// TIA Portal V20 export
FUNCTION_BLOCK "CallEquipment"   // FB72, LAD
TITLE = CallEquipment
// This block includes all general functions, checks and logik that is needed in the entire unit. E.g. general releases and system wide functionalities like air, pressure and power handling as well as general reaction to events.
// stored: IsIECCheckEnabled true, MemoryReserve 100, Namespace Unit1.Em8, SetENOAutomatically true
   VAR_INPUT
      ZoneOperationEnable { ExternalWritable := 'False'} : "LWONIK_typeSafetyZoneManualOperation";
   END_VAR
   VAR_IN_OUT
      unitStatus : "LAF_typeUnitStatus";   // Current unit status o be used in this EM
      emFeedback : "LUC_typeEmFeedback";   // Feedback of the EM to the Unit
      unitAlarmDB : "LAF_typeAlarms";   // Summarized EM Alarms for the Unit
   END_VAR
   VAR
      InstHipotThicknessSequence { ExternalWritable := 'False'} : "Unit1.Em8.Sequence_1_HipotThickness";
      InstHipotThicknessRnRSequence { S7_SetPoint := 'True'} : "Unit1.Em8.Sequence_10_GuageRnR";
      instHipotThicknessHomeJob1 { ExternalWritable := 'False'} : "LAF_SelectJob";
      instHipotThicknessLoadJob2 { ExternalWritable := 'False'} : "LAF_SelectJob";
      instHipotThicknessInspectionJob3 { ExternalWritable := 'False'} : "LAF_SelectJob";
      instHipotThicknessUnloadJob4 { ExternalWritable := 'False'} : "LAF_SelectJob";
      instGRnR_HipotThicknessLoad_Job2 { S7_SetPoint := 'True'} : "LAF_SelectJob";
      instGRnR_HipotThicknessInspection_Job3 { S7_SetPoint := 'True'} : "LAF_SelectJob";
      instGRnR_HipotThicknessUnload_Job4 { S7_SetPoint := 'True'} : "LAF_SelectJob";
      instCmHipotThicknessSafetyPin { ExternalWritable := 'False'} : "LBC_DigitalSignalCn";
      instCmHipotThicknessJRDetect { ExternalWritable := 'False'} : "LBC_DigitalSignalCn";
      instCmThicknessAxisZ { ExternalWritable := 'False'} : "LBC_Axis64Pos_TecPlcCn";
      instCmHipotThinknessStageLiftFrontUpDown { ExternalWritable := 'False'} : "LBC_TwoWayActuatorCn";
      instCmHipotThinknessStageLiftRearUpDown { ExternalWritable := 'False'} : "LBC_TwoWayActuatorCn";
      instCmHipotTabContactorBwdFwd { ExternalWritable := 'False'} : "LBC_TwoWayActuatorCn";
      instCmHipotTabContactorLeftOpenClose { ExternalWritable := 'False'} : "LBC_TwoWayActuatorCn";
      instCmHipotTabContactorRightOpenClose { ExternalWritable := 'False'} : "LBC_TwoWayActuatorCn";
      instCmHipotThinknessStageLiftAllUpDown { ExternalWritable := 'False'} : "LBC_TwoWayActuatorCn";
      instCmHipotControl { ExternalWritable := 'False'} : "LER_IRCheck_BT5525";
      instCmThicknessControl { ExternalWritable := 'False'} : "LER_Thickness";
      instCmHipotThicknessServoPress { ExternalWritable := 'False'} : "LER_ServoPress";
      instInterlockThicknessAxisZ { ExternalWritable := 'False'} : "LER_Axis64Pos_InterlockSummary";
      instLDrv701ControlThicknessAxisZ { ExternalWritable := 'False'} : "LDrvSafe_SinaTlg701Control";   // Drive Telegram Function Library
      instLDrv701StatusThicknessAxisZ { ExternalWritable := 'False'} : "LDrvSafe_SinaTlg701Status";   // Drive Telegram Function Library
      instHipotThicknessPressHistory { ExternalWritable := 'False'} : "LER_ServoPressHistory";
      instHipotHistory { ExternalWritable := 'False'} : "LER_hipotHistory";
      instThicknessHistory { ExternalWritable := 'False'} : "LER_thicknessHistory";
      instManageAlarms { ExternalWritable := 'False'} : "LAF_ManageAlarms";
      instEventsPFE { ExternalWritable := 'False'} : "Unit1.Em8.EventsPFE";
      statUnitStatus { ExternalWritable := 'False'} : "LAF_typeUnitStatus";   // Unit Status that is used in this project
      statSlmStatus { ExternalWritable := 'False'} : Struct
         running : Bool;
         powerOff : Bool;
      END_STRUCT;
      statAllBrakeTest { ExternalWritable := 'False'} : "LER_typeBrakeTestUnitCommands";
      statPartData { ExternalWritable := 'False'} : "LER_typePartData";
      statDataDelete { ExternalWritable := 'False'} : "LER_typePartData";
      statHistoryDeleteData_press { ExternalWritable := 'False'} : "LER_typeServoPressHistory";
      statHistoryDeleteData_hipot { ExternalWritable := 'False'} : "LER_typeHipotHistory";
      statHistoryDeleteData_thickness { ExternalWritable := 'False'} : "LER_typeThicknessHistory";
      "statHistoryDeleteData_thicknessR&R" { ExternalWritable := 'False'} : "LER_typeThicknessHistory_R&R";
      statRoutingOk { ExternalWritable := 'False'} : Array[0..99] of Bool;
      statRoutingNok { ExternalWritable := 'False'} : Array[0..99] of Bool;
      statTonTime { ExternalWritable := 'False'} : Array[0..999] of TON_TIME;
      statTofTime { ExternalWritable := 'False'} : Array[0..9] of TOF_TIME;
      statPulse { ExternalWritable := 'False'} : Array[0..999] of Bool;
      statGaugeRnR { ExternalWritable := 'False'} : Struct
         currentCount : Int;
         processCount : Int;
         Ongoing : Bool;
         Complete : Bool;
      END_STRUCT;
      statEnableManualCmds { ExternalWritable := 'False'} : Bool;
      statNomalMode { ExternalWritable := 'False'} : Bool;
      "*** Interlock Axis ***" : Bool;
      ThicknessAxisZ_Jog { S7_SetPoint := 'True'} : Array[0..2] of "LER_Axis_Jog";
      ThicknessAxisZ_interlock { S7_SetPoint := 'True'} : Array[0..10] of "LER_Axis_Absolute";
      ThicknessAxisZ_IntPos : Array[0..9] of Struct
         "Int" : Array[1..10] of Bool;
      END_STRUCT;
      ThicknessAxisZ_IntHome : Array[0..9] of Bool;
      ThicknessAxisZ_PosAbsolute : Array[0..10] of Bool;
      ThicknessAxisZ_Home { S7_SetPoint := 'True'} : "LER_Axis_Homing";
      "*** Interlock TwoWay ***" { S7_SetPoint := 'True'} : "LER_Axis_Homing";
      instCmHipotThinknessStageLiftFrontUpDownInterlock { S7_SetPoint := 'True'} : Array[0..2] of "LER_Actuator";
      instCmHipotThinknessStageLiftRearUpDownInterlock { S7_SetPoint := 'True'} : Array[0..2] of "LER_Actuator";
      instCmHipotTabContactorBwdFwdInterlock { S7_SetPoint := 'True'} : Array[0..2] of "LER_Actuator";
      instCmHipotTabContactorLeftOpenCloseInterlock { S7_SetPoint := 'True'} : Array[0..2] of "LER_Actuator";
      instCmHipotTabContactorRightOpenCloseInterlock { S7_SetPoint := 'True'} : Array[0..2] of "LER_Actuator";
      instCmHipotThinknessStageLiftAllUpDownInterlock { S7_SetPoint := 'True'} : Array[0..2] of "LER_Actuator";
      HipotThinknessStageLiftFrontUpDown_Inpos : Array[0..2] of Struct
         "Int" : Array[1..10] of Bool;
      END_STRUCT;
      HipotThinknessStageLiftRearUpDown_Inpos : Array[0..2] of Struct
         "Int" : Array[1..10] of Bool;
      END_STRUCT;
      HipotTabContactorBwdFwd_Inpos : Array[0..2] of Struct
         "Int" : Array[1..10] of Bool;
      END_STRUCT;
      HipotTabContactorLeftOpenClose_Inpos : Array[0..2] of Struct
         "Int" : Array[1..10] of Bool;
      END_STRUCT;
      HipotTabContactorRightOpenClose_Inpos : Array[0..2] of Struct
         "Int" : Array[1..10] of Bool;
      END_STRUCT;
      HipotThinknessStageLiftAllUpDown_Inpos : Array[0..2] of Struct
         "Int" : Array[1..10] of Bool;
      END_STRUCT;
      citi_Ptrig : Array[0..20] of Bool;
      citiTon : Array[0..20] of TON_TIME;
      citi : Time;
      citiTest : Array[0..20] of Bool;
      instPFERecipe { S7_SetPoint := 'True'} : "Unit1.Em8.EventsPFE_Recipe";
   END_VAR
   VAR_TEMP
      tempRET_VAL : Array[0..99] of Int;
      tempScInProduction : Bool;   // Mode Production and StateComplete
      tempScNoProduction : Bool;   // Mode Manual and StateComplete
      tempPlaceReq : Bool;   // Request placing to TRPnPRight
      tempInspecReq : Bool;
      tempPickReq : Bool;   // Request Pick to TRPnPRight
   END_VAR
   VAR CONSTANT
      delayTime : Time := T#3s;
      TRUE : Bool := TRUE;
      FALSE : Bool;
      NO_JOB : DInt;
      MIN_POSITION_NUMBER : SInt;
      INIT_POSITION_NUMBER : SInt := -1;
   END_VAR
   VAR_TEMP   // added for the SCL form of the ladder/FBD networks
      _w1 : Bool;
      _w2 : Bool;
      _w3 : Bool;
      _w4 : Bool;
      _w5 : Bool;
      _w6 : Bool;
      _w7 : Bool;
      _w8 : Bool;
      _w9 : Bool;
      _w10 : Bool;
      _w11 : Bool;
      _w12 : Bool;
   END_VAR
BEGIN

REGION Network 1: BLOCK INFO HEADER
   // (company) / (C) Copyright (year)
   // ---------------------------------------------------------------------------------
   // Title:                             (Title of this block)
   // Comment/Function: (that is implemented in the block)
   // Library/Family:           (that the source is dedicated to)
   // Author:                        (department / person in charge / contact)
   // Target System:          (test system with FW version)
   // Engineering:              TIA Portal (SW version)
   // Restrictions:               (OB types, etc.)
   // Requirements:           (hardware, technological package, etc.)
   // ---------------------------------------------------------------------------------
   // Change log table:
   // Version          | Date             | Signature      | Expert in charge  | Changes applied ------------------------|----------------------|-------------------------|--------------------------------|-----------------------
   // 001.000.000 | yyyy-mm-dd | 0x00000000 | (name of expert) | First released version
END_REGION

REGION Network 2: DESCRIPTION
   // This is a template block provided by the Automation Framework. It can be used to create an own project.
   // The Block Info Header is prepared to put in your own data.
   // Description of the block could be added here and the docu created by Code2Docu.
END_REGION

REGION Network 3: Simulation
   // If simulation is active on a global level, inherit this status and set simulation active in this unit also. Information is written to DB ControlNodes, from where it is distributed to the equipmemt modules.
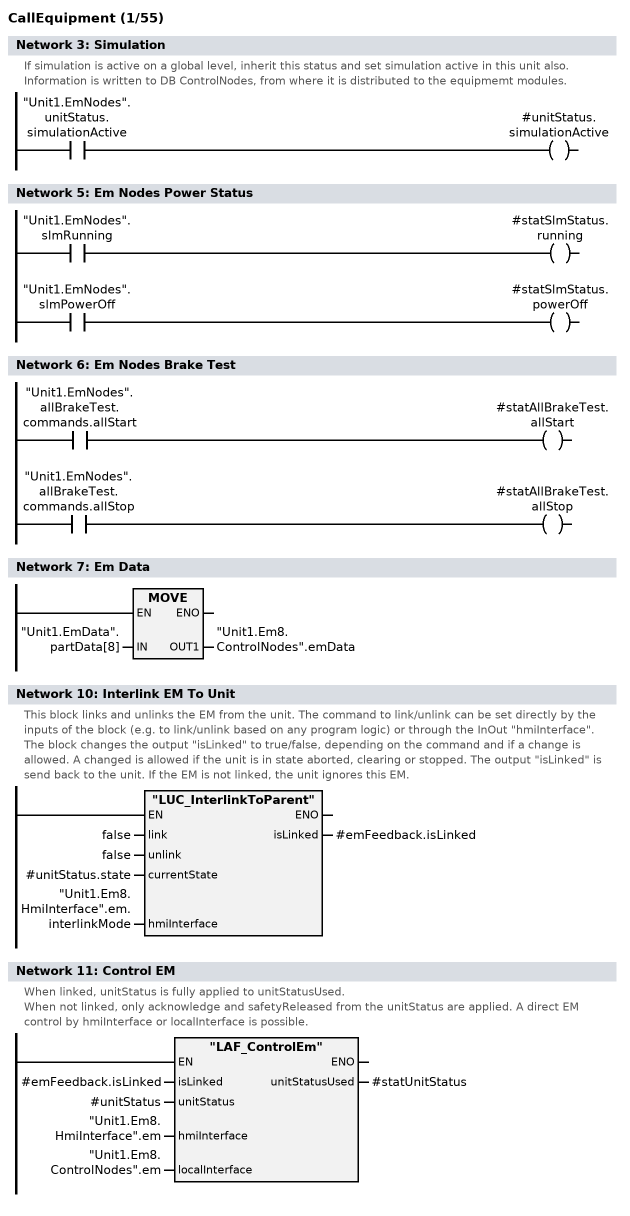
   RUNG wire#powerrail
      Contact( "Unit1.EmNodes".unitStatus.simulationActive )
      Coil( #unitStatus.simulationActive )
   END_RUNG
   // the same network as SCL:
   #unitStatus.simulationActive := "Unit1.EmNodes".unitStatus.simulationActive;
END_REGION

REGION Network 4: ******************** Unit Input ********************
END_REGION

REGION Network 5: Em Nodes Power Status
   RUNG wire#powerrail
      Contact( "Unit1.EmNodes".slmRunning )
      Coil( #statSlmStatus.running )
   END_RUNG
   RUNG wire#powerrail
      Contact( "Unit1.EmNodes".slmPowerOff )
      Coil( #statSlmStatus.powerOff )
   END_RUNG
   // the same network as SCL:
   #statSlmStatus.running := "Unit1.EmNodes".slmRunning;
   #statSlmStatus.powerOff := "Unit1.EmNodes".slmPowerOff;
END_REGION

REGION Network 6: Em Nodes Brake Test
   RUNG wire#powerrail
      Contact( "Unit1.EmNodes".allBrakeTest.commands.allStart )
      Coil( #statAllBrakeTest.allStart )
   END_RUNG
   RUNG wire#powerrail
      Contact( "Unit1.EmNodes".allBrakeTest.commands.allStop )
      Coil( #statAllBrakeTest.allStop )
   END_RUNG
   // the same network as SCL:
   #statAllBrakeTest.allStart := "Unit1.EmNodes".allBrakeTest.commands.allStart;
   #statAllBrakeTest.allStop := "Unit1.EmNodes".allBrakeTest.commands.allStop;
END_REGION

REGION Network 7: Em Data
   RUNG wire#powerrail
      Move(in := "Unit1.EmData".partData[8], out1 => "Unit1.Em8.ControlNodes".emData)
   END_RUNG
   // the same network as SCL:
   "Unit1.Em8.ControlNodes".emData := "Unit1.EmData".partData[8];
END_REGION

REGION Network 9: ******************** Equipment Control ********************
END_REGION

REGION Network 10: Interlink EM To Unit
   // This block links and unlinks the EM from the unit. The command to link/unlink can be set directly by the inputs of the block (e.g. to link/unlink based on any program logic) or through the InOut "hmiInterface". The block changes the output "isLinked" to true/false, depending on the command and if a change is allowed. A changed is allowed if the unit is in state aborted, clearing or stopped. The output "isLinked" is send back to the unit. If the EM is not linked, the unit ignores this EM.
   RUNG wire#powerrail
      "LUC_InterlinkToParent"(link := false, unlink := false, currentState := #unitStatus.state, hmiInterface := "Unit1.Em8.HmiInterface".em.interlinkMode, isLinked => #emFeedback.isLinked)
   END_RUNG
   // the same network as SCL:
   "LUC_InterlinkToParent"(link := false,
                           unlink := false,
                           currentState := #unitStatus.state,
                           hmiInterface := "Unit1.Em8.HmiInterface".em.interlinkMode,
                           isLinked => #emFeedback.isLinked);
END_REGION

REGION Network 11: Control EM
   // When linked, unitStatus is fully applied to unitStatusUsed.
   // When not linked, only acknowledge and safetyReleased from the unitStatus are applied. A direct EM control by hmiInterface or localInterface is possible.
   RUNG wire#powerrail
      "LAF_ControlEm"(isLinked := #emFeedback.isLinked, unitStatus := #unitStatus, hmiInterface := "Unit1.Em8.HmiInterface".em, localInterface := "Unit1.Em8.ControlNodes".em, unitStatusUsed => #statUnitStatus)
   END_RUNG
   // the same network as SCL:
   "LAF_ControlEm"(isLinked := #emFeedback.isLinked,
                   unitStatus := #unitStatus,
                   hmiInterface := "Unit1.Em8.HmiInterface".em,
                   localInterface := "Unit1.Em8.ControlNodes".em,
                   unitStatusUsed => #statUnitStatus);
END_REGION

REGION Network 12: EnableManualCmds
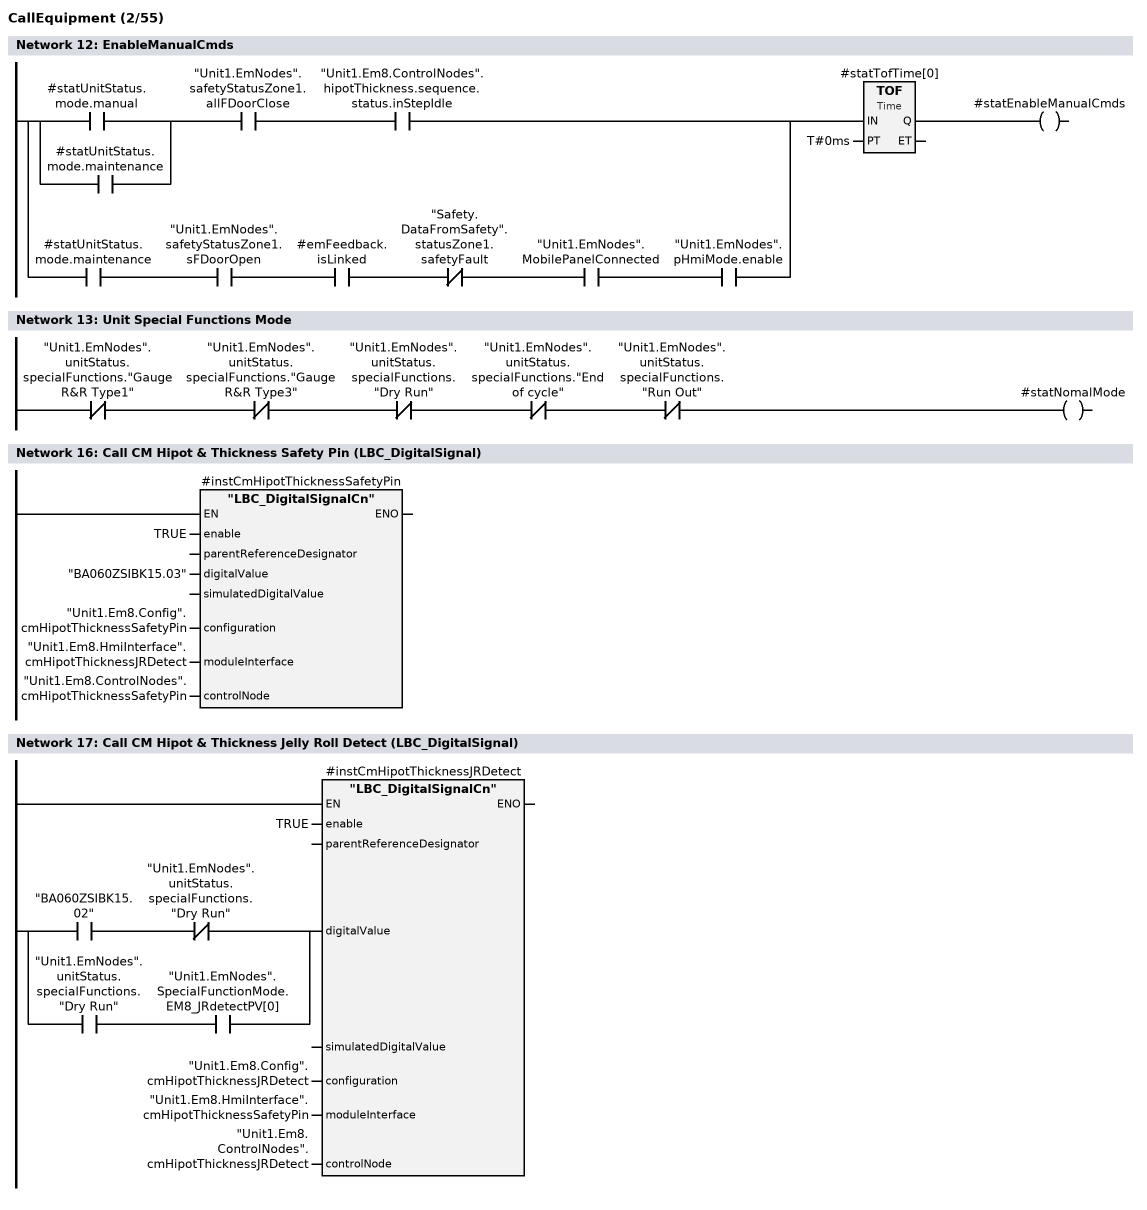
   RUNG wire#powerrail
      Contact( #statUnitStatus.mode.manual )
      wire#w1
      Contact( "Unit1.EmNodes".safetyStatusZone1.allFDoorClose )
      Contact( "Unit1.Em8.ControlNodes".hipotThickness.sequence.status.inStepIdle )
      wire#w2
      { S7_Templates := "time_type := Time" } #statTofTime[0].TOF(pt := T#0ms, et =>)
      Coil( #statEnableManualCmds )
   END_RUNG
   RUNG wire#powerrail
      Contact( #statUnitStatus.mode.maintenance )
   END_RUNG wire#w1
   RUNG wire#powerrail
      Contact( #statUnitStatus.mode.maintenance )
      Contact( "Unit1.EmNodes".safetyStatusZone1.sFDoorOpen )
      Contact( #emFeedback.isLinked )
      I_Contact( "Safety.DataFromSafety".statusZone1.safetyFault )
      Contact( "Unit1.EmNodes".MobilePanelConnected )
      Contact( "Unit1.EmNodes".pHmiMode.enable )
   END_RUNG wire#w2
   // the same network as SCL:
   #statTofTime[0].TOF(IN := ((#statUnitStatus.mode.manual OR #statUnitStatus.mode.maintenance) AND "Unit1.EmNodes".safetyStatusZone1.allFDoorClose AND "Unit1.Em8.ControlNodes".hipotThickness.sequence.status.inStepIdle) OR (#statUnitStatus.mode.maintenance AND "Unit1.EmNodes".safetyStatusZone1.sFDoorOpen AND #emFeedback.isLinked AND NOT "Safety.DataFromSafety".statusZone1.safetyFault AND "Unit1.EmNodes".MobilePanelConnected AND "Unit1.EmNodes".pHmiMode.enable),
                       PT := T#0ms);
   #statEnableManualCmds := #statTofTime[0].Q;
END_REGION

REGION Network 13: Unit Special Functions Mode
   RUNG wire#powerrail
      I_Contact( "Unit1.EmNodes".unitStatus.specialFunctions."Gauge R&R Type1" )
      I_Contact( "Unit1.EmNodes".unitStatus.specialFunctions."Gauge R&R Type3" )
      I_Contact( "Unit1.EmNodes".unitStatus.specialFunctions."Dry Run" )
      I_Contact( "Unit1.EmNodes".unitStatus.specialFunctions."End of cycle" )
      I_Contact( "Unit1.EmNodes".unitStatus.specialFunctions."Run Out" )
      Coil( #statNomalMode )
   END_RUNG
   // the same network as SCL:
   #statNomalMode := NOT "Unit1.EmNodes".unitStatus.specialFunctions."Gauge R&R Type1" AND NOT "Unit1.EmNodes".unitStatus.specialFunctions."Gauge R&R Type3" AND NOT "Unit1.EmNodes".unitStatus.specialFunctions."Dry Run" AND NOT "Unit1.EmNodes".unitStatus.specialFunctions."End of cycle" AND NOT "Unit1.EmNodes".unitStatus.specialFunctions."Run Out";
END_REGION

REGION Network 15: ******************** Control Modules (Sensors) ********************
   // Call control modules that are sensors before the em logic (jobs and sequence), so that the latest value is used in the logic.
END_REGION

REGION Network 16: Call CM Hipot & Thickness Safety Pin (LBC_DigitalSignal)
   RUNG wire#powerrail
      #instCmHipotThicknessSafetyPin(enable := TRUE, parentReferenceDesignator :=, digitalValue := "BA060ZSIBK15.03", simulatedDigitalValue :=, configuration := "Unit1.Em8.Config".cmHipotThicknessSafetyPin, moduleInterface := "Unit1.Em8.HmiInterface".cmHipotThicknessJRDetect, controlNode := "Unit1.Em8.ControlNodes".cmHipotThicknessSafetyPin)
   END_RUNG
   // the same network as SCL:
   #instCmHipotThicknessSafetyPin(enable := TRUE,   // "LBC_DigitalSignalCn"
                           digitalValue := "BA060ZSIBK15.03",
                           configuration := "Unit1.Em8.Config".cmHipotThicknessSafetyPin,
                           moduleInterface := "Unit1.Em8.HmiInterface".cmHipotThicknessJRDetect,
                           controlNode := "Unit1.Em8.ControlNodes".cmHipotThicknessSafetyPin);
END_REGION

REGION Network 17: Call CM Hipot & Thickness Jelly Roll Detect (LBC_DigitalSignal)
   RUNG wire#powerrail
      #instCmHipotThicknessJRDetect(digitalValue := wire#w1, enable := TRUE, parentReferenceDesignator :=, simulatedDigitalValue :=, configuration := "Unit1.Em8.Config".cmHipotThicknessJRDetect, moduleInterface := "Unit1.Em8.HmiInterface".cmHipotThicknessSafetyPin, controlNode := "Unit1.Em8.ControlNodes".cmHipotThicknessJRDetect)
   END_RUNG
   RUNG wire#powerrail
      Contact( "BA060ZSIBK15.02" )
      I_Contact( "Unit1.EmNodes".unitStatus.specialFunctions."Dry Run" )
   END_RUNG wire#w1
   RUNG wire#powerrail
      Contact( "Unit1.EmNodes".unitStatus.specialFunctions."Dry Run" )
      Contact( "Unit1.EmNodes".SpecialFunctionMode.EM8_JRdetectPV[0] )
   END_RUNG wire#w1
   // the same network as SCL:
   #instCmHipotThicknessJRDetect(enable := TRUE,   // "LBC_DigitalSignalCn"
                           digitalValue := ("BA060ZSIBK15.02" AND NOT "Unit1.EmNodes".unitStatus.specialFunctions."Dry Run") OR ("Unit1.EmNodes".unitStatus.specialFunctions."Dry Run" AND "Unit1.EmNodes".SpecialFunctionMode.EM8_JRdetectPV[0]),
                           configuration := "Unit1.Em8.Config".cmHipotThicknessJRDetect,
                           moduleInterface := "Unit1.Em8.HmiInterface".cmHipotThicknessSafetyPin,
                           controlNode := "Unit1.Em8.ControlNodes".cmHipotThicknessJRDetect);
END_REGION

REGION Network 19: ******************** Equipment Logic ********************
END_REGION

REGION Network 20: Map Unit Status To Sequence Status
   // This block maps the unit status to the seuqnce status. Thus, it controls the sequence depending on the unit status. E.g. it sets the sequence to automatic when the unit state is in productions. This blocks work perfectly with the sequences provided in the AF. 
   // This typed block (MapUnitStatusToSequence) could be adjusted to specific application requirements or if other, user-defined sequences are used.
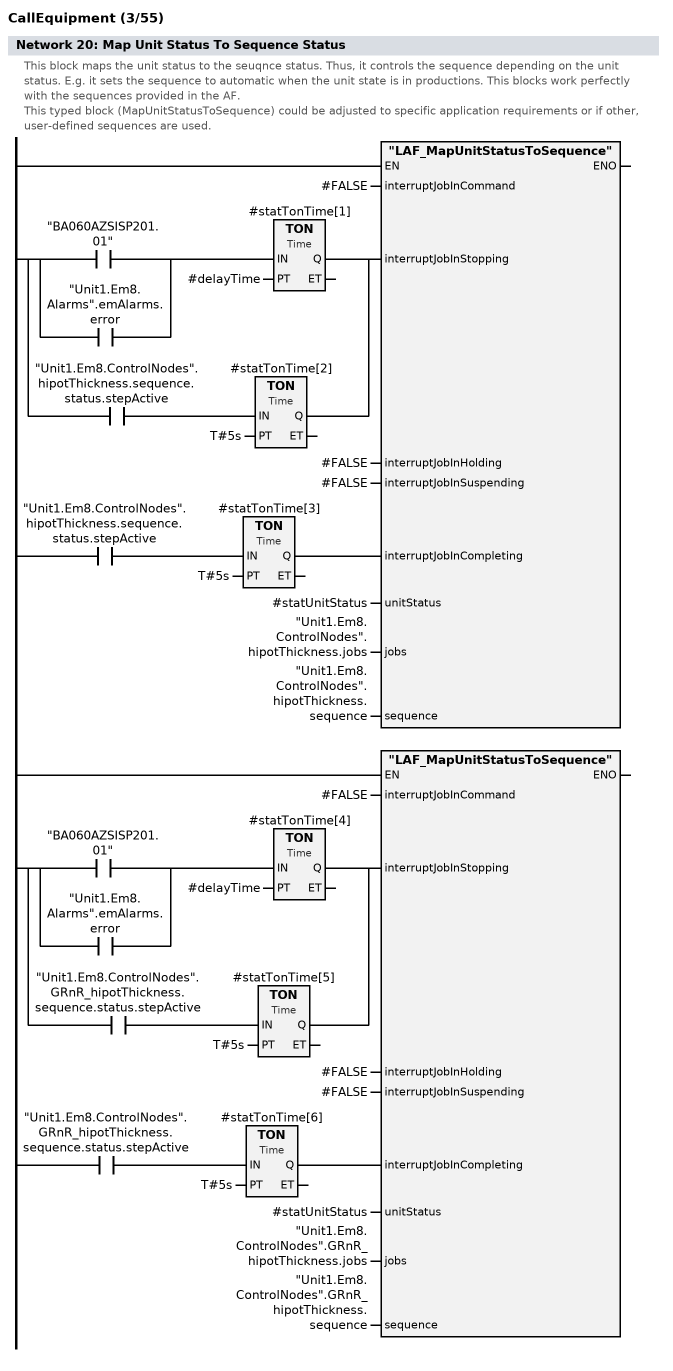
   RUNG wire#powerrail
      "LAF_MapUnitStatusToSequence"(interruptJobInStopping := wire#w2, interruptJobInCompleting := wire#w3, interruptJobInCommand := #FALSE, interruptJobInHolding := #FALSE, interruptJobInSuspending := #FALSE, unitStatus := #statUnitStatus, jobs := "Unit1.Em8.ControlNodes".hipotThickness.jobs, sequence := "Unit1.Em8.ControlNodes".hipotThickness.sequence)
   END_RUNG
   RUNG wire#powerrail
      Contact( "BA060AZSISP201.01" )
      wire#w1
      { S7_Templates := "time_type := Time" } #statTonTime[1].TON(pt := #delayTime, et =>)
   END_RUNG wire#w2
   RUNG wire#powerrail
      Contact( "Unit1.Em8.Alarms".emAlarms.error )
   END_RUNG wire#w1
   RUNG wire#powerrail
      Contact( "Unit1.Em8.ControlNodes".hipotThickness.sequence.status.stepActive )
      { S7_Templates := "time_type := Time" } #statTonTime[2].TON(pt := T#5s, et =>)
   END_RUNG wire#w2
   RUNG wire#powerrail
      Contact( "Unit1.Em8.ControlNodes".hipotThickness.sequence.status.stepActive )
      { S7_Templates := "time_type := Time" } #statTonTime[3].TON(pt := T#5s, et =>)
   END_RUNG wire#w3
   RUNG wire#powerrail
      "LAF_MapUnitStatusToSequence"(interruptJobInStopping := wire#w5, interruptJobInCompleting := wire#w6, interruptJobInCommand := #FALSE, interruptJobInHolding := #FALSE, interruptJobInSuspending := #FALSE, unitStatus := #statUnitStatus, jobs := "Unit1.Em8.ControlNodes".GRnR_hipotThickness.jobs, sequence := "Unit1.Em8.ControlNodes".GRnR_hipotThickness.sequence)
   END_RUNG
   RUNG wire#powerrail
      Contact( "BA060AZSISP201.01" )
      wire#w4
      { S7_Templates := "time_type := Time" } #statTonTime[4].TON(pt := #delayTime, et =>)
   END_RUNG wire#w5
   RUNG wire#powerrail
      Contact( "Unit1.Em8.Alarms".emAlarms.error )
   END_RUNG wire#w4
   RUNG wire#powerrail
      Contact( "Unit1.Em8.ControlNodes".GRnR_hipotThickness.sequence.status.stepActive )
      { S7_Templates := "time_type := Time" } #statTonTime[5].TON(pt := T#5s, et =>)
   END_RUNG wire#w5
   RUNG wire#powerrail
      Contact( "Unit1.Em8.ControlNodes".GRnR_hipotThickness.sequence.status.stepActive )
      { S7_Templates := "time_type := Time" } #statTonTime[6].TON(pt := T#5s, et =>)
   END_RUNG wire#w6
   // the same network as SCL:
   #statTonTime[1].TON(IN := "BA060AZSISP201.01" OR "Unit1.Em8.Alarms".emAlarms.error, PT := #delayTime);
   #_w1 := #statTonTime[1].Q;
   #statTonTime[2].TON(IN := "Unit1.Em8.ControlNodes".hipotThickness.sequence.status.stepActive, PT := T#5s);
   #_w2 := #_w1 OR #statTonTime[2].Q;
   #statTonTime[3].TON(IN := "Unit1.Em8.ControlNodes".hipotThickness.sequence.status.stepActive, PT := T#5s);
   "LAF_MapUnitStatusToSequence"(interruptJobInCommand := #FALSE,
                           interruptJobInStopping := #_w2,
                           interruptJobInHolding := #FALSE,
                           interruptJobInSuspending := #FALSE,
                           interruptJobInCompleting := #statTonTime[3].Q,
                           unitStatus := #statUnitStatus,
                           jobs := "Unit1.Em8.ControlNodes".hipotThickness.jobs,
                           sequence := "Unit1.Em8.ControlNodes".hipotThickness.sequence);
   #statTonTime[4].TON(IN := "BA060AZSISP201.01" OR "Unit1.Em8.Alarms".emAlarms.error, PT := #delayTime);
   #_w3 := #statTonTime[4].Q;
   #statTonTime[5].TON(IN := "Unit1.Em8.ControlNodes".GRnR_hipotThickness.sequence.status.stepActive,
                       PT := T#5s);
   #_w4 := #_w3 OR #statTonTime[5].Q;
   #statTonTime[6].TON(IN := "Unit1.Em8.ControlNodes".GRnR_hipotThickness.sequence.status.stepActive,
                       PT := T#5s);
   "LAF_MapUnitStatusToSequence"(interruptJobInCommand := #FALSE,
                           interruptJobInStopping := #_w4,
                           interruptJobInHolding := #FALSE,
                           interruptJobInSuspending := #FALSE,
                           interruptJobInCompleting := #statTonTime[6].Q,
                           unitStatus := #statUnitStatus,
                           jobs := "Unit1.Em8.ControlNodes".GRnR_hipotThickness.jobs,
                           sequence := "Unit1.Em8.ControlNodes".GRnR_hipotThickness.sequence);
END_REGION

REGION Network 21: {SpecialFunction} DryRun
   // _."BA060ZSIBK15.02"
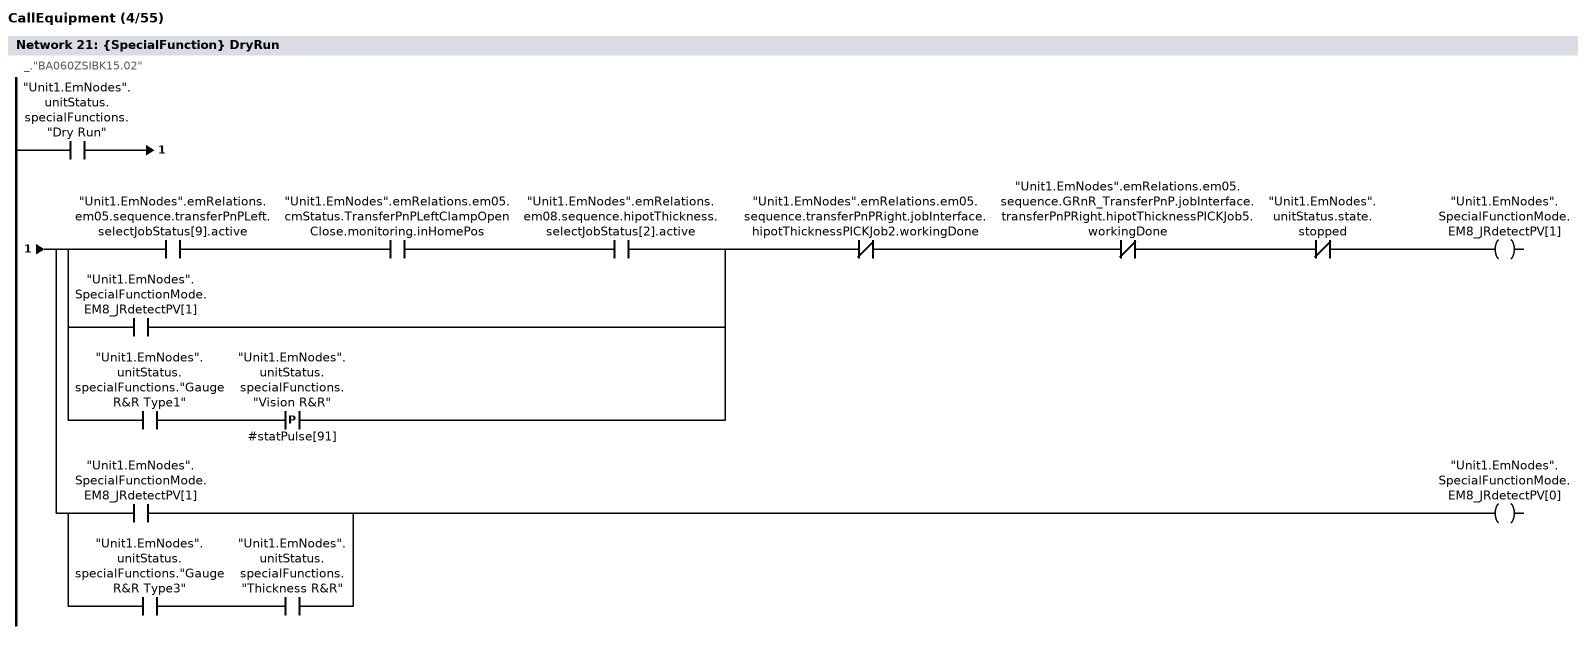
   RUNG wire#powerrail
      Contact( "Unit1.EmNodes".unitStatus.specialFunctions."Dry Run" )
      wire#w1
      Contact( "Unit1.EmNodes".emRelations.em05.sequence.transferPnPLeft.selectJobStatus[9].active )
      Contact( "Unit1.EmNodes".emRelations.em05.cmStatus.TransferPnPLeftClampOpenClose.monitoring.inHomePos )
      Contact( "Unit1.EmNodes".emRelations.em08.sequence.hipotThickness.selectJobStatus[2].active )
      wire#w2
      I_Contact( "Unit1.EmNodes".emRelations.em05.sequence.transferPnPRight.jobInterface.hipotThicknessPICKJob2.workingDone )
      I_Contact( "Unit1.EmNodes".emRelations.em05.sequence.GRnR_TransferPnP.jobInterface.transferPnPRight.hipotThicknessPICKJob5.workingDone )
      I_Contact( "Unit1.EmNodes".unitStatus.state.stopped )
      Coil( "Unit1.EmNodes".SpecialFunctionMode.EM8_JRdetectPV[1] )
   END_RUNG
   RUNG wire#w1
      Contact( "Unit1.EmNodes".SpecialFunctionMode.EM8_JRdetectPV[1] )
   END_RUNG wire#w2
   RUNG wire#w1
      Contact( "Unit1.EmNodes".unitStatus.specialFunctions."Gauge R&R Type1" )
      P_Contact(operand := "Unit1.EmNodes".unitStatus.specialFunctions."Vision R&R", bit := #statPulse[91])
   END_RUNG wire#w2
   RUNG wire#w1
      Contact( "Unit1.EmNodes".SpecialFunctionMode.EM8_JRdetectPV[1] )
      wire#w3
      Coil( "Unit1.EmNodes".SpecialFunctionMode.EM8_JRdetectPV[0] )
   END_RUNG
   RUNG wire#w1
      Contact( "Unit1.EmNodes".unitStatus.specialFunctions."Gauge R&R Type3" )
      Contact( "Unit1.EmNodes".unitStatus.specialFunctions."Thickness R&R" )
   END_RUNG wire#w3
   // the same network as SCL:
   #_w1 := "Unit1.EmNodes".unitStatus.specialFunctions."Dry Run" AND "Unit1.EmNodes".unitStatus.specialFunctions."Gauge R&R Type1" AND "Unit1.EmNodes".unitStatus.specialFunctions."Vision R&R" AND NOT #statPulse[91];   // rising edge of "Unit1.EmNodes".unitStatus.specialFunctions."Vision R&R"
   #statPulse[91] := "Unit1.EmNodes".unitStatus.specialFunctions."Vision R&R";
   "Unit1.EmNodes".SpecialFunctionMode.EM8_JRdetectPV[1] := (("Unit1.EmNodes".unitStatus.specialFunctions."Dry Run" AND (("Unit1.EmNodes".emRelations.em05.sequence.transferPnPLeft.selectJobStatus[9].active AND "Unit1.EmNodes".emRelations.em05.cmStatus.TransferPnPLeftClampOpenClose.monitoring.inHomePos AND "Unit1.EmNodes".emRelations.em08.sequence.hipotThickness.selectJobStatus[2].active) OR "Unit1.EmNodes".SpecialFunctionMode.EM8_JRdetectPV[1])) OR #_w1) AND NOT "Unit1.EmNodes".emRelations.em05.sequence.transferPnPRight.jobInterface.hipotThicknessPICKJob2.workingDone AND NOT "Unit1.EmNodes".emRelations.em05.sequence.GRnR_TransferPnP.jobInterface.transferPnPRight.hipotThicknessPICKJob5.workingDone AND NOT "Unit1.EmNodes".unitStatus.state.stopped;
   "Unit1.EmNodes".SpecialFunctionMode.EM8_JRdetectPV[0] := "Unit1.EmNodes".unitStatus.specialFunctions."Dry Run" AND ("Unit1.EmNodes".SpecialFunctionMode.EM8_JRdetectPV[1] OR ("Unit1.EmNodes".unitStatus.specialFunctions."Gauge R&R Type3" AND "Unit1.EmNodes".unitStatus.specialFunctions."Thickness R&R"));
END_REGION

REGION Network 23: [Job] Hipot & Thickness Select Job
   // Configure here when the jobs of the sequence should be started. More jobs could be added.
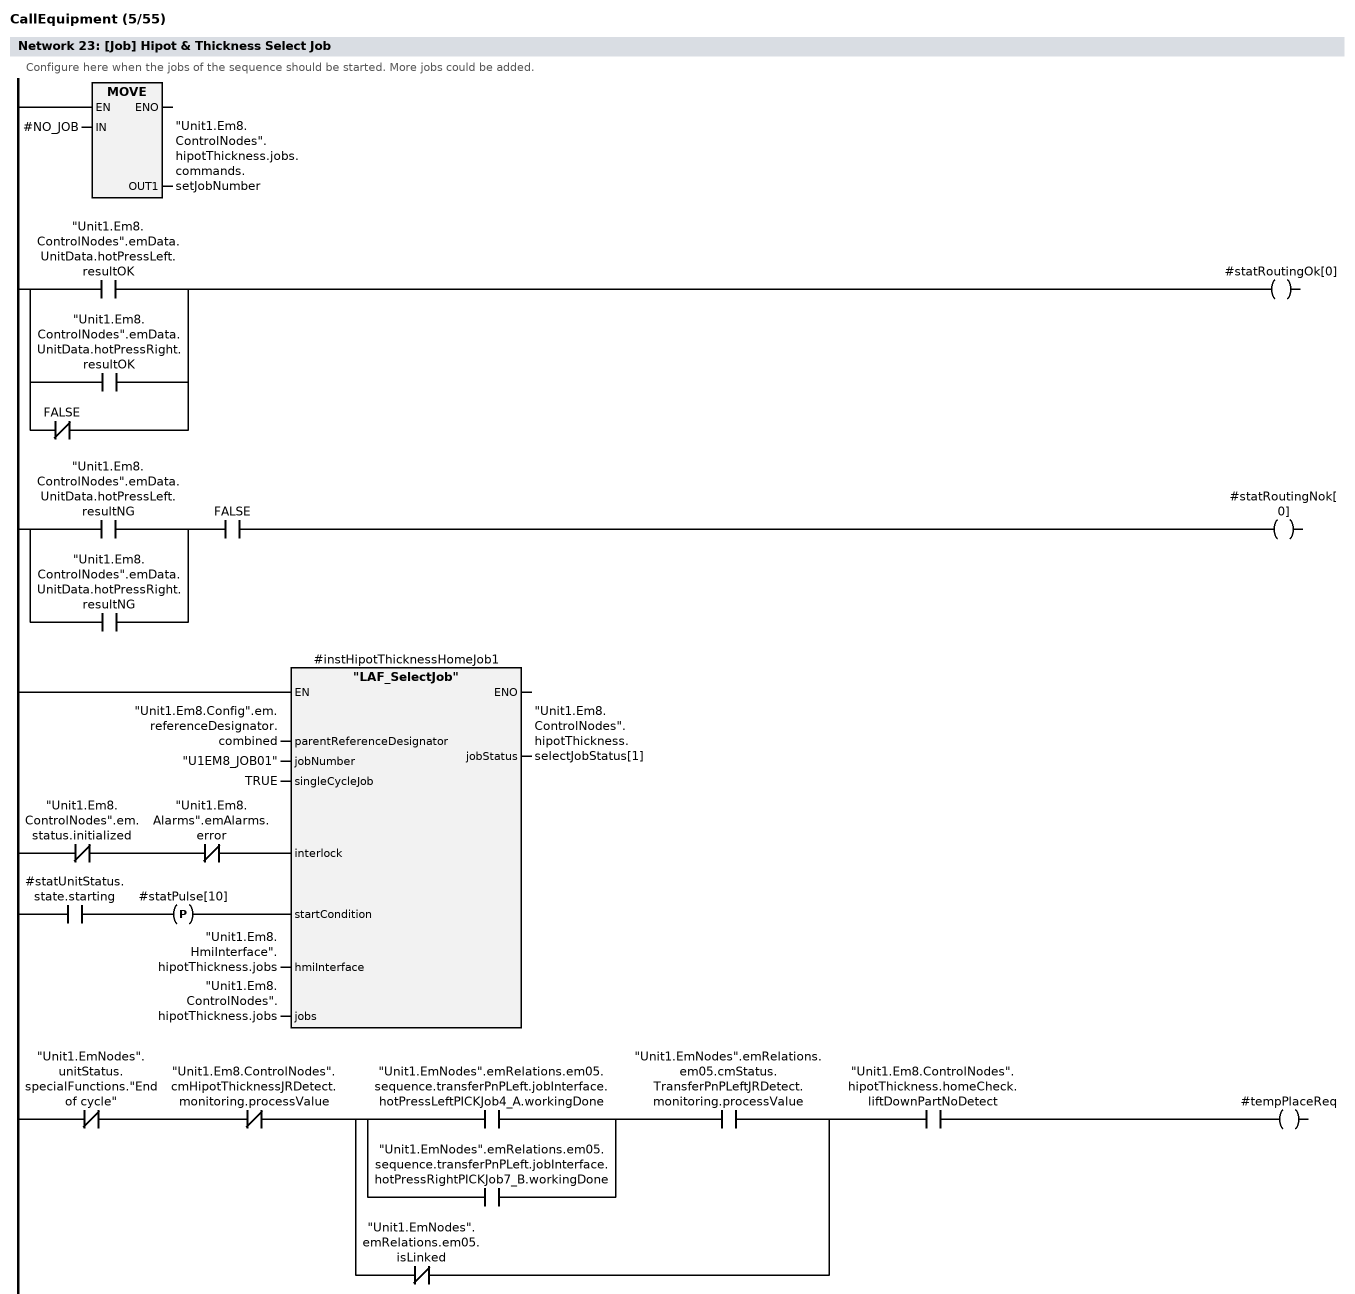
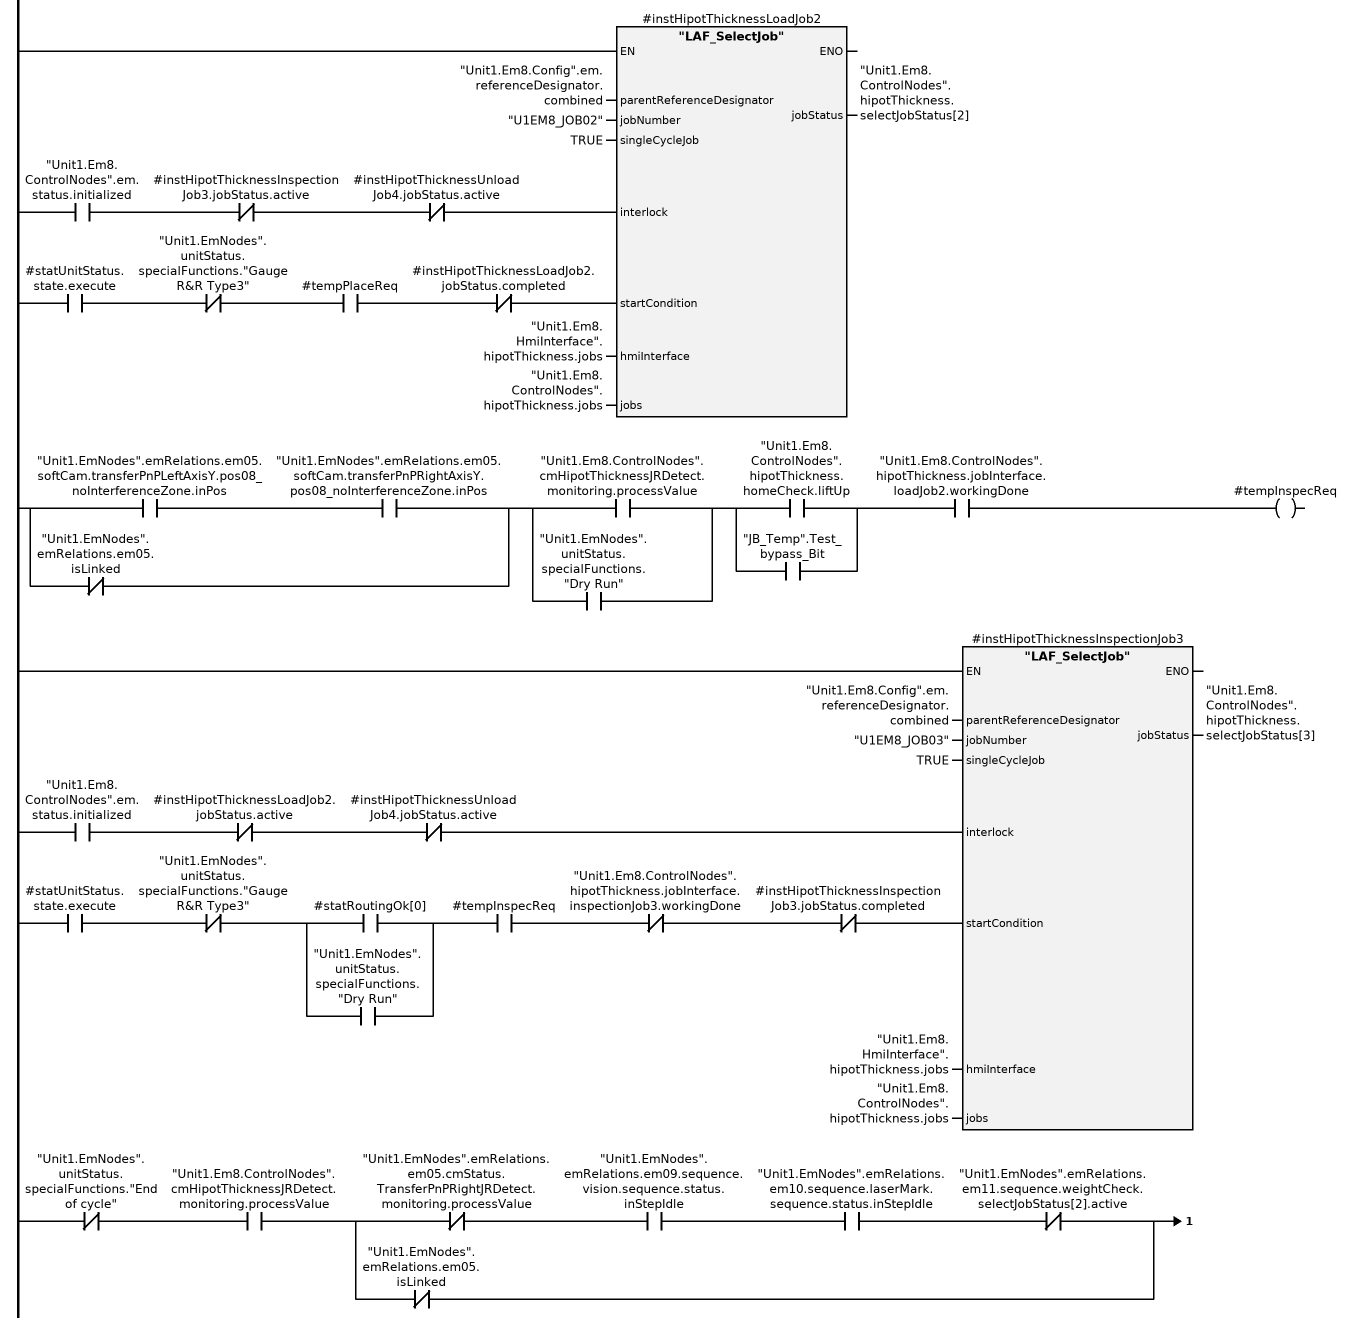
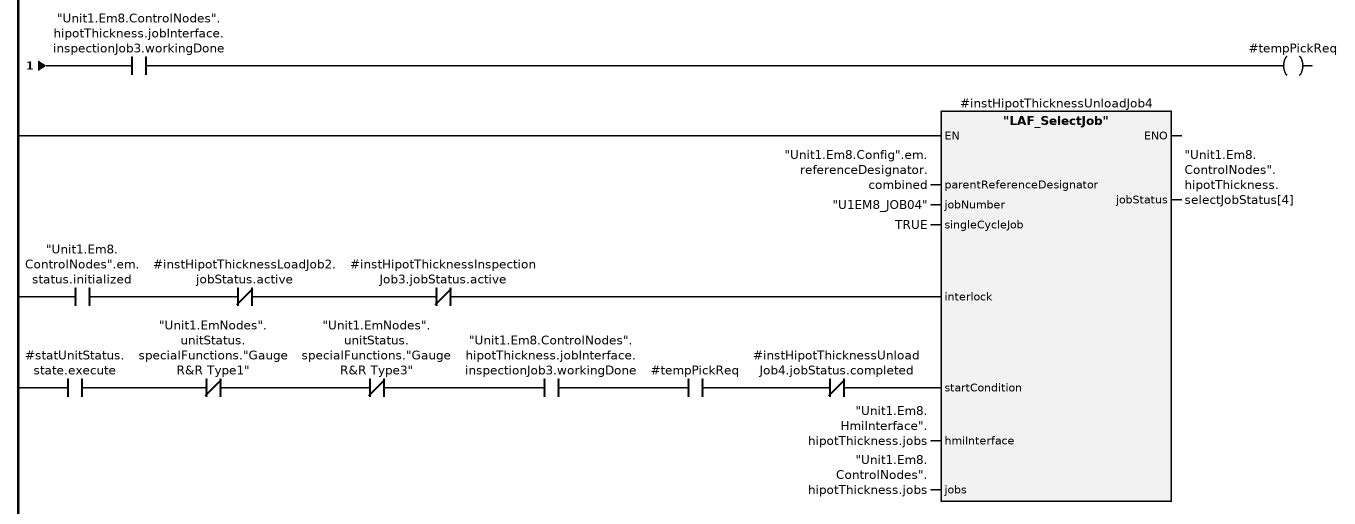
   RUNG wire#powerrail
      Move(in := #NO_JOB, out1 => "Unit1.Em8.ControlNodes".hipotThickness.jobs.commands.setJobNumber)
   END_RUNG
   RUNG wire#powerrail
      Contact( "Unit1.Em8.ControlNodes".emData.UnitData.hotPressLeft.resultOK )
      wire#w1
      Coil( #statRoutingOk[0] )
   END_RUNG
   RUNG wire#powerrail
      Contact( "Unit1.Em8.ControlNodes".emData.UnitData.hotPressRight.resultOK )
   END_RUNG wire#w1
   RUNG wire#powerrail
      I_Contact( FALSE )
   END_RUNG wire#w1
   RUNG wire#powerrail
      Contact( "Unit1.Em8.ControlNodes".emData.UnitData.hotPressLeft.resultNG )
      wire#w2
      Contact( FALSE )
      Coil( #statRoutingNok[0] )
   END_RUNG
   RUNG wire#powerrail
      Contact( "Unit1.Em8.ControlNodes".emData.UnitData.hotPressRight.resultNG )
   END_RUNG wire#w2
   RUNG wire#powerrail
      #instHipotThicknessHomeJob1(interlock := wire#w3, startCondition := wire#w4, parentReferenceDesignator := "Unit1.Em8.Config".em.referenceDesignator.combined, jobNumber := "U1EM8_JOB01", singleCycleJob := TRUE, hmiInterface := "Unit1.Em8.HmiInterface".hipotThickness.jobs, jobs := "Unit1.Em8.ControlNodes".hipotThickness.jobs, jobStatus => "Unit1.Em8.ControlNodes".hipotThickness.selectJobStatus[1])
   END_RUNG
   RUNG wire#powerrail
      I_Contact( "Unit1.Em8.ControlNodes".em.status.initialized )
      I_Contact( "Unit1.Em8.Alarms".emAlarms.error )
   END_RUNG wire#w3
   RUNG wire#powerrail
      Contact( #statUnitStatus.state.starting )
      P_Trig( #statPulse[10] )
   END_RUNG wire#w4
   RUNG wire#powerrail
      I_Contact( "Unit1.EmNodes".unitStatus.specialFunctions."End of cycle" )
      I_Contact( "Unit1.Em8.ControlNodes".cmHipotThicknessJRDetect.monitoring.processValue )
      wire#w5
      Contact( "Unit1.EmNodes".emRelations.em05.sequence.transferPnPLeft.jobInterface.hotPressLeftPICKJob4_A.workingDone )
      wire#w6
      Contact( "Unit1.EmNodes".emRelations.em05.cmStatus.TransferPnPLeftJRDetect.monitoring.processValue )
      wire#w7
      Contact( "Unit1.Em8.ControlNodes".hipotThickness.homeCheck.liftDownPartNoDetect )
      Coil( #tempPlaceReq )
   END_RUNG
   RUNG wire#w5
      Contact( "Unit1.EmNodes".emRelations.em05.sequence.transferPnPLeft.jobInterface.hotPressRightPICKJob7_B.workingDone )
   END_RUNG wire#w6
   RUNG wire#w5
      I_Contact( "Unit1.EmNodes".emRelations.em05.isLinked )
   END_RUNG wire#w7
   RUNG wire#powerrail
      #instHipotThicknessLoadJob2(interlock := wire#w8, startCondition := wire#w9, parentReferenceDesignator := "Unit1.Em8.Config".em.referenceDesignator.combined, jobNumber := "U1EM8_JOB02", singleCycleJob := TRUE, hmiInterface := "Unit1.Em8.HmiInterface".hipotThickness.jobs, jobs := "Unit1.Em8.ControlNodes".hipotThickness.jobs, jobStatus => "Unit1.Em8.ControlNodes".hipotThickness.selectJobStatus[2])
   END_RUNG
   RUNG wire#powerrail
      Contact( "Unit1.Em8.ControlNodes".em.status.initialized )
      I_Contact( #instHipotThicknessInspectionJob3.jobStatus.active )
      I_Contact( #instHipotThicknessUnloadJob4.jobStatus.active )
   END_RUNG wire#w8
   RUNG wire#powerrail
      Contact( #statUnitStatus.state.execute )
      I_Contact( "Unit1.EmNodes".unitStatus.specialFunctions."Gauge R&R Type3" )
      Contact( #tempPlaceReq )
      I_Contact( #instHipotThicknessLoadJob2.jobStatus.completed )
   END_RUNG wire#w9
   RUNG wire#powerrail
      Contact( "Unit1.EmNodes".emRelations.em05.softCam.transferPnPLeftAxisY.pos08_noInterferenceZone.inPos )
      Contact( "Unit1.EmNodes".emRelations.em05.softCam.transferPnPRightAxisY.pos08_noInterferenceZone.inPos )
      wire#w10
      Contact( "Unit1.Em8.ControlNodes".cmHipotThicknessJRDetect.monitoring.processValue )
      wire#w11
      Contact( "Unit1.Em8.ControlNodes".hipotThickness.homeCheck.liftUp )
      wire#w12
      Contact( "Unit1.Em8.ControlNodes".hipotThickness.jobInterface.loadJob2.workingDone )
      Coil( #tempInspecReq )
   END_RUNG
   RUNG wire#powerrail
      I_Contact( "Unit1.EmNodes".emRelations.em05.isLinked )
   END_RUNG wire#w10
   RUNG wire#w10
      Contact( "Unit1.EmNodes".unitStatus.specialFunctions."Dry Run" )
   END_RUNG wire#w11
   RUNG wire#w11
      Contact( "JB_Temp".Test_bypass_Bit )
   END_RUNG wire#w12
   RUNG wire#powerrail
      #instHipotThicknessInspectionJob3(interlock := wire#w13, startCondition := wire#w16, parentReferenceDesignator := "Unit1.Em8.Config".em.referenceDesignator.combined, jobNumber := "U1EM8_JOB03", singleCycleJob := TRUE, hmiInterface := "Unit1.Em8.HmiInterface".hipotThickness.jobs, jobs := "Unit1.Em8.ControlNodes".hipotThickness.jobs, jobStatus => "Unit1.Em8.ControlNodes".hipotThickness.selectJobStatus[3])
   END_RUNG
   RUNG wire#powerrail
      Contact( "Unit1.Em8.ControlNodes".em.status.initialized )
      I_Contact( #instHipotThicknessLoadJob2.jobStatus.active )
      I_Contact( #instHipotThicknessUnloadJob4.jobStatus.active )
   END_RUNG wire#w13
   RUNG wire#powerrail
      Contact( #statUnitStatus.state.execute )
      I_Contact( "Unit1.EmNodes".unitStatus.specialFunctions."Gauge R&R Type3" )
      wire#w14
      Contact( #statRoutingOk[0] )
      wire#w15
      Contact( #tempInspecReq )
      I_Contact( "Unit1.Em8.ControlNodes".hipotThickness.jobInterface.inspectionJob3.workingDone )
      I_Contact( #instHipotThicknessInspectionJob3.jobStatus.completed )
   END_RUNG wire#w16
   RUNG wire#w14
      Contact( "Unit1.EmNodes".unitStatus.specialFunctions."Dry Run" )
   END_RUNG wire#w15
   RUNG wire#powerrail
      I_Contact( "Unit1.EmNodes".unitStatus.specialFunctions."End of cycle" )
      Contact( "Unit1.Em8.ControlNodes".cmHipotThicknessJRDetect.monitoring.processValue )
      wire#w17
      I_Contact( "Unit1.EmNodes".emRelations.em05.cmStatus.TransferPnPRightJRDetect.monitoring.processValue )
      Contact( "Unit1.EmNodes".emRelations.em09.sequence.vision.sequence.status.inStepIdle )
      Contact( "Unit1.EmNodes".emRelations.em10.sequence.laserMark.sequence.status.inStepIdle )
      I_Contact( "Unit1.EmNodes".emRelations.em11.sequence.weightCheck.selectJobStatus[2].active )
      wire#w18
      Contact( "Unit1.Em8.ControlNodes".hipotThickness.jobInterface.inspectionJob3.workingDone )
      Coil( #tempPickReq )
   END_RUNG
   RUNG wire#w17
      I_Contact( "Unit1.EmNodes".emRelations.em05.isLinked )
   END_RUNG wire#w18
   RUNG wire#powerrail
      #instHipotThicknessUnloadJob4(interlock := wire#w19, startCondition := wire#w20, parentReferenceDesignator := "Unit1.Em8.Config".em.referenceDesignator.combined, jobNumber := "U1EM8_JOB04", singleCycleJob := TRUE, hmiInterface := "Unit1.Em8.HmiInterface".hipotThickness.jobs, jobs := "Unit1.Em8.ControlNodes".hipotThickness.jobs, jobStatus => "Unit1.Em8.ControlNodes".hipotThickness.selectJobStatus[4])
   END_RUNG
   RUNG wire#powerrail
      Contact( "Unit1.Em8.ControlNodes".em.status.initialized )
      I_Contact( #instHipotThicknessLoadJob2.jobStatus.active )
      I_Contact( #instHipotThicknessInspectionJob3.jobStatus.active )
   END_RUNG wire#w19
   RUNG wire#powerrail
      Contact( #statUnitStatus.state.execute )
      I_Contact( "Unit1.EmNodes".unitStatus.specialFunctions."Gauge R&R Type1" )
      I_Contact( "Unit1.EmNodes".unitStatus.specialFunctions."Gauge R&R Type3" )
      Contact( "Unit1.Em8.ControlNodes".hipotThickness.jobInterface.inspectionJob3.workingDone )
      Contact( #tempPickReq )
      I_Contact( #instHipotThicknessUnloadJob4.jobStatus.completed )
   END_RUNG wire#w20
   // the same network as SCL:
   "Unit1.Em8.ControlNodes".hipotThickness.jobs.commands.setJobNumber := #NO_JOB;
   #statRoutingOk[0] := "Unit1.Em8.ControlNodes".emData.UnitData.hotPressLeft.resultOK OR "Unit1.Em8.ControlNodes".emData.UnitData.hotPressRight.resultOK OR NOT FALSE;
   #statRoutingNok[0] := ("Unit1.Em8.ControlNodes".emData.UnitData.hotPressLeft.resultNG OR "Unit1.Em8.ControlNodes".emData.UnitData.hotPressRight.resultNG) AND FALSE;
   #_w1 := #statUnitStatus.state.starting AND NOT #statPulse[10];   // rising edge
   #statPulse[10] := #statUnitStatus.state.starting;
   #instHipotThicknessHomeJob1(parentReferenceDesignator := "Unit1.Em8.Config".em.referenceDesignator.combined,   // "LAF_SelectJob"
                           jobNumber := "U1EM8_JOB01",
                           singleCycleJob := TRUE,
                           interlock := NOT "Unit1.Em8.ControlNodes".em.status.initialized AND NOT "Unit1.Em8.Alarms".emAlarms.error,
                           startCondition := #_w1,
                           hmiInterface := "Unit1.Em8.HmiInterface".hipotThickness.jobs,
                           jobs := "Unit1.Em8.ControlNodes".hipotThickness.jobs,
                           jobStatus => "Unit1.Em8.ControlNodes".hipotThickness.selectJobStatus[1]);
   #tempPlaceReq := NOT "Unit1.EmNodes".unitStatus.specialFunctions."End of cycle" AND NOT "Unit1.Em8.ControlNodes".cmHipotThicknessJRDetect.monitoring.processValue AND ((("Unit1.EmNodes".emRelations.em05.sequence.transferPnPLeft.jobInterface.hotPressLeftPICKJob4_A.workingDone OR "Unit1.EmNodes".emRelations.em05.sequence.transferPnPLeft.jobInterface.hotPressRightPICKJob7_B.workingDone) AND "Unit1.EmNodes".emRelations.em05.cmStatus.TransferPnPLeftJRDetect.monitoring.processValue) OR NOT "Unit1.EmNodes".emRelations.em05.isLinked) AND "Unit1.Em8.ControlNodes".hipotThickness.homeCheck.liftDownPartNoDetect;
   #instHipotThicknessLoadJob2(parentReferenceDesignator := "Unit1.Em8.Config".em.referenceDesignator.combined,   // "LAF_SelectJob"
                           jobNumber := "U1EM8_JOB02",
                           singleCycleJob := TRUE,
                           interlock := "Unit1.Em8.ControlNodes".em.status.initialized AND NOT #instHipotThicknessInspectionJob3.jobStatus.active AND NOT #instHipotThicknessUnloadJob4.jobStatus.active,
                           startCondition := #statUnitStatus.state.execute AND NOT "Unit1.EmNodes".unitStatus.specialFunctions."Gauge R&R Type3" AND #tempPlaceReq AND NOT #instHipotThicknessLoadJob2.jobStatus.completed,
                           hmiInterface := "Unit1.Em8.HmiInterface".hipotThickness.jobs,
                           jobs := "Unit1.Em8.ControlNodes".hipotThickness.jobs,
                           jobStatus => "Unit1.Em8.ControlNodes".hipotThickness.selectJobStatus[2]);
   #tempInspecReq := (("Unit1.EmNodes".emRelations.em05.softCam.transferPnPLeftAxisY.pos08_noInterferenceZone.inPos AND "Unit1.EmNodes".emRelations.em05.softCam.transferPnPRightAxisY.pos08_noInterferenceZone.inPos) OR NOT "Unit1.EmNodes".emRelations.em05.isLinked) AND ("Unit1.Em8.ControlNodes".cmHipotThicknessJRDetect.monitoring.processValue OR "Unit1.EmNodes".unitStatus.specialFunctions."Dry Run") AND ("Unit1.Em8.ControlNodes".hipotThickness.homeCheck.liftUp OR "JB_Temp".Test_bypass_Bit) AND "Unit1.Em8.ControlNodes".hipotThickness.jobInterface.loadJob2.workingDone;
   #instHipotThicknessInspectionJob3(parentReferenceDesignator := "Unit1.Em8.Config".em.referenceDesignator.combined,   // "LAF_SelectJob"
                           jobNumber := "U1EM8_JOB03",
                           singleCycleJob := TRUE,
                           interlock := "Unit1.Em8.ControlNodes".em.status.initialized AND NOT #instHipotThicknessLoadJob2.jobStatus.active AND NOT #instHipotThicknessUnloadJob4.jobStatus.active,
                           startCondition := #statUnitStatus.state.execute AND NOT "Unit1.EmNodes".unitStatus.specialFunctions."Gauge R&R Type3" AND (#statRoutingOk[0] OR "Unit1.EmNodes".unitStatus.specialFunctions."Dry Run") AND #tempInspecReq AND NOT "Unit1.Em8.ControlNodes".hipotThickness.jobInterface.inspectionJob3.workingDone AND NOT #instHipotThicknessInspectionJob3.jobStatus.completed,
                           hmiInterface := "Unit1.Em8.HmiInterface".hipotThickness.jobs,
                           jobs := "Unit1.Em8.ControlNodes".hipotThickness.jobs,
                           jobStatus => "Unit1.Em8.ControlNodes".hipotThickness.selectJobStatus[3]);
   #tempPickReq := NOT "Unit1.EmNodes".unitStatus.specialFunctions."End of cycle" AND "Unit1.Em8.ControlNodes".cmHipotThicknessJRDetect.monitoring.processValue AND ((NOT "Unit1.EmNodes".emRelations.em05.cmStatus.TransferPnPRightJRDetect.monitoring.processValue AND "Unit1.EmNodes".emRelations.em09.sequence.vision.sequence.status.inStepIdle AND "Unit1.EmNodes".emRelations.em10.sequence.laserMark.sequence.status.inStepIdle AND NOT "Unit1.EmNodes".emRelations.em11.sequence.weightCheck.selectJobStatus[2].active) OR NOT "Unit1.EmNodes".emRelations.em05.isLinked) AND "Unit1.Em8.ControlNodes".hipotThickness.jobInterface.inspectionJob3.workingDone;
   #instHipotThicknessUnloadJob4(parentReferenceDesignator := "Unit1.Em8.Config".em.referenceDesignator.combined,   // "LAF_SelectJob"
                           jobNumber := "U1EM8_JOB04",
                           singleCycleJob := TRUE,
                           interlock := "Unit1.Em8.ControlNodes".em.status.initialized AND NOT #instHipotThicknessLoadJob2.jobStatus.active AND NOT #instHipotThicknessInspectionJob3.jobStatus.active,
                           startCondition := #statUnitStatus.state.execute AND NOT "Unit1.EmNodes".unitStatus.specialFunctions."Gauge R&R Type1" AND NOT "Unit1.EmNodes".unitStatus.specialFunctions."Gauge R&R Type3" AND "Unit1.Em8.ControlNodes".hipotThickness.jobInterface.inspectionJob3.workingDone AND #tempPickReq AND NOT #instHipotThicknessUnloadJob4.jobStatus.completed,
                           hmiInterface := "Unit1.Em8.HmiInterface".hipotThickness.jobs,
                           jobs := "Unit1.Em8.ControlNodes".hipotThickness.jobs,
                           jobStatus => "Unit1.Em8.ControlNodes".hipotThickness.selectJobStatus[4]);
END_REGION

REGION Network 24: Hipot & Thickness Job Interface [Loading]
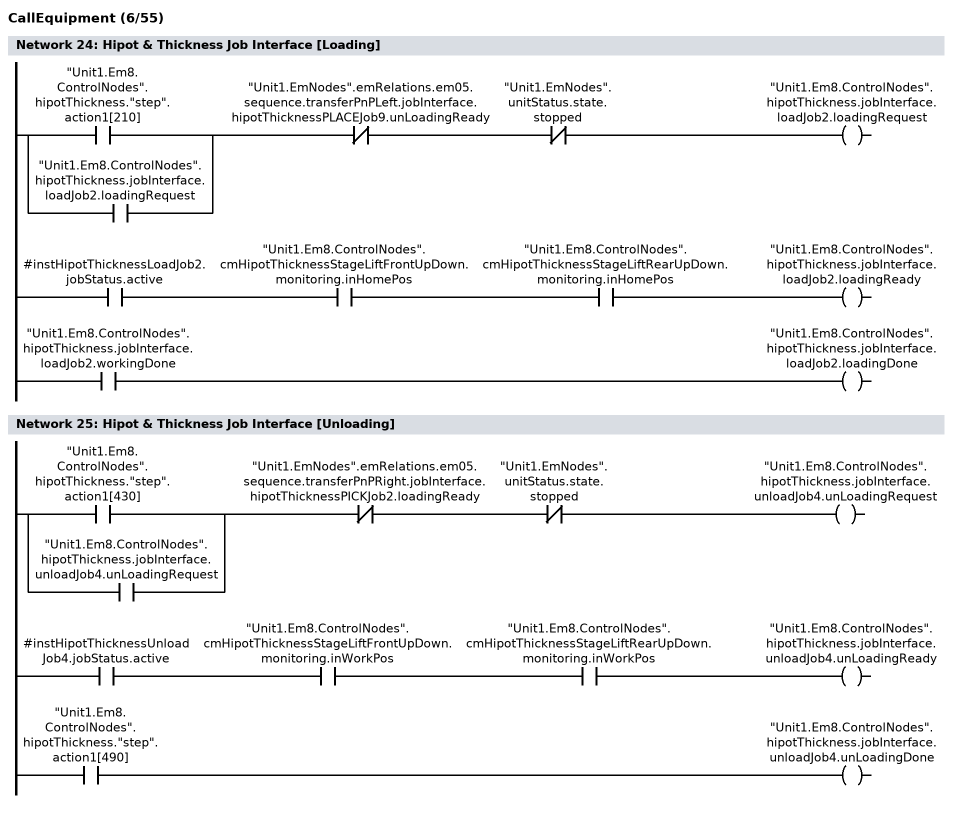
   RUNG wire#powerrail
      Contact( "Unit1.Em8.ControlNodes".hipotThickness."step".action1[210] )
      wire#w1
      I_Contact( "Unit1.EmNodes".emRelations.em05.sequence.transferPnPLeft.jobInterface.hipotThicknessPLACEJob9.unLoadingReady )
      I_Contact( "Unit1.EmNodes".unitStatus.state.stopped )
      Coil( "Unit1.Em8.ControlNodes".hipotThickness.jobInterface.loadJob2.loadingRequest )
   END_RUNG
   RUNG wire#powerrail
      Contact( "Unit1.Em8.ControlNodes".hipotThickness.jobInterface.loadJob2.loadingRequest )
   END_RUNG wire#w1
   RUNG wire#powerrail
      Contact( #instHipotThicknessLoadJob2.jobStatus.active )
      Contact( "Unit1.Em8.ControlNodes".cmHipotThicknessStageLiftFrontUpDown.monitoring.inHomePos )
      Contact( "Unit1.Em8.ControlNodes".cmHipotThicknessStageLiftRearUpDown.monitoring.inHomePos )
      Coil( "Unit1.Em8.ControlNodes".hipotThickness.jobInterface.loadJob2.loadingReady )
   END_RUNG
   RUNG wire#powerrail
      Contact( "Unit1.Em8.ControlNodes".hipotThickness.jobInterface.loadJob2.workingDone )
      Coil( "Unit1.Em8.ControlNodes".hipotThickness.jobInterface.loadJob2.loadingDone )
   END_RUNG
   // the same network as SCL:
   "Unit1.Em8.ControlNodes".hipotThickness.jobInterface.loadJob2.loadingRequest := ("Unit1.Em8.ControlNodes".hipotThickness."step".action1[210] OR "Unit1.Em8.ControlNodes".hipotThickness.jobInterface.loadJob2.loadingRequest) AND NOT "Unit1.EmNodes".emRelations.em05.sequence.transferPnPLeft.jobInterface.hipotThicknessPLACEJob9.unLoadingReady AND NOT "Unit1.EmNodes".unitStatus.state.stopped;
   "Unit1.Em8.ControlNodes".hipotThickness.jobInterface.loadJob2.loadingReady := #instHipotThicknessLoadJob2.jobStatus.active AND "Unit1.Em8.ControlNodes".cmHipotThicknessStageLiftFrontUpDown.monitoring.inHomePos AND "Unit1.Em8.ControlNodes".cmHipotThicknessStageLiftRearUpDown.monitoring.inHomePos;
   "Unit1.Em8.ControlNodes".hipotThickness.jobInterface.loadJob2.loadingDone := "Unit1.Em8.ControlNodes".hipotThickness.jobInterface.loadJob2.workingDone;
END_REGION

REGION Network 25: Hipot & Thickness Job Interface [Unloading]
   RUNG wire#powerrail
      Contact( "Unit1.Em8.ControlNodes".hipotThickness."step".action1[430] )
      wire#w1
      I_Contact( "Unit1.EmNodes".emRelations.em05.sequence.transferPnPRight.jobInterface.hipotThicknessPICKJob2.loadingReady )
      I_Contact( "Unit1.EmNodes".unitStatus.state.stopped )
      Coil( "Unit1.Em8.ControlNodes".hipotThickness.jobInterface.unloadJob4.unLoadingRequest )
   END_RUNG
   RUNG wire#powerrail
      Contact( "Unit1.Em8.ControlNodes".hipotThickness.jobInterface.unloadJob4.unLoadingRequest )
   END_RUNG wire#w1
   RUNG wire#powerrail
      Contact( #instHipotThicknessUnloadJob4.jobStatus.active )
      Contact( "Unit1.Em8.ControlNodes".cmHipotThicknessStageLiftFrontUpDown.monitoring.inWorkPos )
      Contact( "Unit1.Em8.ControlNodes".cmHipotThicknessStageLiftRearUpDown.monitoring.inWorkPos )
      Coil( "Unit1.Em8.ControlNodes".hipotThickness.jobInterface.unloadJob4.unLoadingReady )
   END_RUNG
   RUNG wire#powerrail
      Contact( "Unit1.Em8.ControlNodes".hipotThickness."step".action1[490] )
      Coil( "Unit1.Em8.ControlNodes".hipotThickness.jobInterface.unloadJob4.unLoadingDone )
   END_RUNG
   // the same network as SCL:
   "Unit1.Em8.ControlNodes".hipotThickness.jobInterface.unloadJob4.unLoadingRequest := ("Unit1.Em8.ControlNodes".hipotThickness."step".action1[430] OR "Unit1.Em8.ControlNodes".hipotThickness.jobInterface.unloadJob4.unLoadingRequest) AND NOT "Unit1.EmNodes".emRelations.em05.sequence.transferPnPRight.jobInterface.hipotThicknessPICKJob2.loadingReady AND NOT "Unit1.EmNodes".unitStatus.state.stopped;
   "Unit1.Em8.ControlNodes".hipotThickness.jobInterface.unloadJob4.unLoadingReady := #instHipotThicknessUnloadJob4.jobStatus.active AND "Unit1.Em8.ControlNodes".cmHipotThicknessStageLiftFrontUpDown.monitoring.inWorkPos AND "Unit1.Em8.ControlNodes".cmHipotThicknessStageLiftRearUpDown.monitoring.inWorkPos;
   "Unit1.Em8.ControlNodes".hipotThickness.jobInterface.unloadJob4.unLoadingDone := "Unit1.Em8.ControlNodes".hipotThickness."step".action1[490];
END_REGION

REGION Network 26: Hipot & Thickness Job Interface Working Done
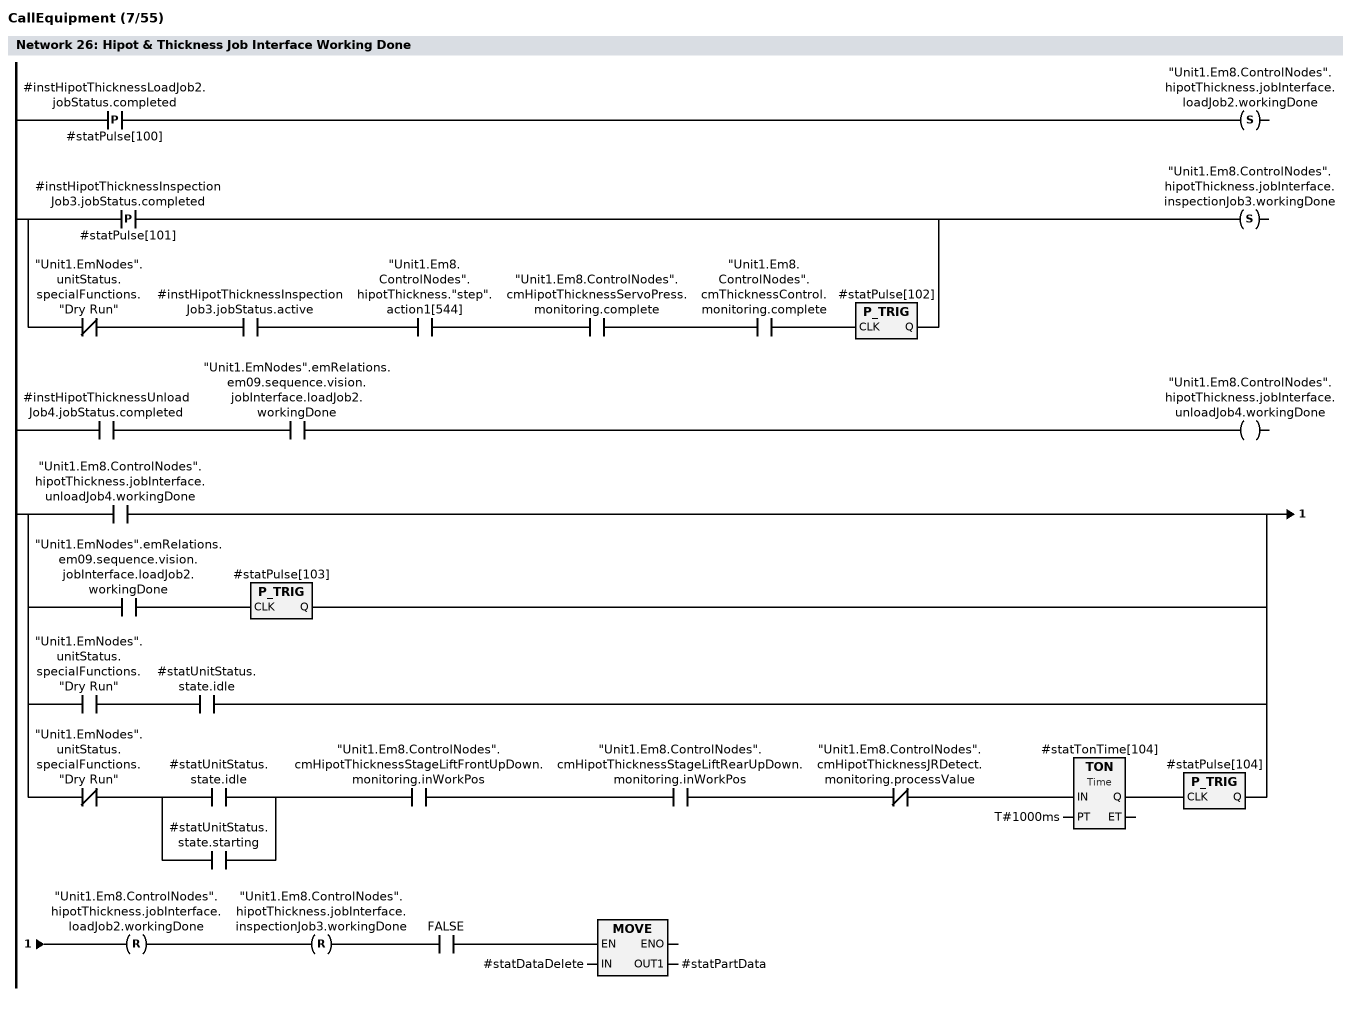
   RUNG wire#powerrail
      P_Contact(operand := #instHipotThicknessLoadJob2.jobStatus.completed, bit := #statPulse[100])
      S_Coil( "Unit1.Em8.ControlNodes".hipotThickness.jobInterface.loadJob2.workingDone )
   END_RUNG
   RUNG wire#powerrail
      P_Contact(operand := #instHipotThicknessInspectionJob3.jobStatus.completed, bit := #statPulse[101])
      wire#w1
      S_Coil( "Unit1.Em8.ControlNodes".hipotThickness.jobInterface.inspectionJob3.workingDone )
   END_RUNG
   RUNG wire#powerrail
      I_Contact( "Unit1.EmNodes".unitStatus.specialFunctions."Dry Run" )
      Contact( #instHipotThicknessInspectionJob3.jobStatus.active )
      Contact( "Unit1.Em8.ControlNodes".hipotThickness."step".action1[544] )
      Contact( "Unit1.Em8.ControlNodes".cmHipotThicknessServoPress.monitoring.complete )
      Contact( "Unit1.Em8.ControlNodes".cmThicknessControl.monitoring.complete )
      P_Trig( #statPulse[102] )
   END_RUNG wire#w1
   RUNG wire#powerrail
      Contact( #instHipotThicknessUnloadJob4.jobStatus.completed )
      Contact( "Unit1.EmNodes".emRelations.em09.sequence.vision.jobInterface.loadJob2.workingDone )
      Coil( "Unit1.Em8.ControlNodes".hipotThickness.jobInterface.unloadJob4.workingDone )
   END_RUNG
   RUNG wire#powerrail
      Contact( "Unit1.Em8.ControlNodes".hipotThickness.jobInterface.unloadJob4.workingDone )
      wire#w2
      R_Coil( "Unit1.Em8.ControlNodes".hipotThickness.jobInterface.loadJob2.workingDone )
      R_Coil( "Unit1.Em8.ControlNodes".hipotThickness.jobInterface.inspectionJob3.workingDone )
      Contact( FALSE )
      Move(in := #statDataDelete, out1 => #statPartData)
   END_RUNG
   RUNG wire#powerrail
      Contact( "Unit1.EmNodes".emRelations.em09.sequence.vision.jobInterface.loadJob2.workingDone )
      P_Trig( #statPulse[103] )
   END_RUNG wire#w2
   RUNG wire#powerrail
      Contact( "Unit1.EmNodes".unitStatus.specialFunctions."Dry Run" )
      Contact( #statUnitStatus.state.idle )
   END_RUNG wire#w2
   RUNG wire#powerrail
      I_Contact( "Unit1.EmNodes".unitStatus.specialFunctions."Dry Run" )
      wire#w3
      Contact( #statUnitStatus.state.idle )
      wire#w4
      Contact( "Unit1.Em8.ControlNodes".cmHipotThicknessStageLiftFrontUpDown.monitoring.inWorkPos )
      Contact( "Unit1.Em8.ControlNodes".cmHipotThicknessStageLiftRearUpDown.monitoring.inWorkPos )
      I_Contact( "Unit1.Em8.ControlNodes".cmHipotThicknessJRDetect.monitoring.processValue )
      { S7_Templates := "time_type := Time" } #statTonTime[104].TON(pt := T#1000ms, et =>)
      P_Trig( #statPulse[104] )
   END_RUNG wire#w2
   RUNG wire#w3
      Contact( #statUnitStatus.state.starting )
   END_RUNG wire#w4
   // the same network as SCL:
   #_w1 := #instHipotThicknessLoadJob2.jobStatus.completed AND NOT #statPulse[100];   // rising edge of #instHipotThicknessLoadJob2.jobStatus.completed
   #statPulse[100] := #instHipotThicknessLoadJob2.jobStatus.completed;
   IF #_w1 THEN "Unit1.Em8.ControlNodes".hipotThickness.jobInterface.loadJob2.workingDone := TRUE; END_IF;
   #_w2 := #instHipotThicknessInspectionJob3.jobStatus.completed AND NOT #statPulse[101];   // rising edge of #instHipotThicknessInspectionJob3.jobStatus.completed
   #statPulse[101] := #instHipotThicknessInspectionJob3.jobStatus.completed;
   #_w3 := NOT "Unit1.EmNodes".unitStatus.specialFunctions."Dry Run" AND #instHipotThicknessInspectionJob3.jobStatus.active AND "Unit1.Em8.ControlNodes".hipotThickness."step".action1[544] AND "Unit1.Em8.ControlNodes".cmHipotThicknessServoPress.monitoring.complete AND "Unit1.Em8.ControlNodes".cmThicknessControl.monitoring.complete;
   #_w4 := #_w3 AND NOT #statPulse[102];   // rising edge
   #statPulse[102] := #_w3;
   IF #_w2 OR #_w4 THEN
       "Unit1.Em8.ControlNodes".hipotThickness.jobInterface.inspectionJob3.workingDone := TRUE;
   END_IF;
   "Unit1.Em8.ControlNodes".hipotThickness.jobInterface.unloadJob4.workingDone := #instHipotThicknessUnloadJob4.jobStatus.completed AND "Unit1.EmNodes".emRelations.em09.sequence.vision.jobInterface.loadJob2.workingDone;
   #_w5 := "Unit1.EmNodes".emRelations.em09.sequence.vision.jobInterface.loadJob2.workingDone AND NOT #statPulse[103];   // rising edge
   #statPulse[103] := "Unit1.EmNodes".emRelations.em09.sequence.vision.jobInterface.loadJob2.workingDone;
   #statTonTime[104].TON(IN := NOT "Unit1.EmNodes".unitStatus.specialFunctions."Dry Run" AND (#statUnitStatus.state.idle OR #statUnitStatus.state.starting) AND "Unit1.Em8.ControlNodes".cmHipotThicknessStageLiftFrontUpDown.monitoring.inWorkPos AND "Unit1.Em8.ControlNodes".cmHipotThicknessStageLiftRearUpDown.monitoring.inWorkPos AND NOT "Unit1.Em8.ControlNodes".cmHipotThicknessJRDetect.monitoring.processValue,
                         PT := T#1000ms);
   #_w6 := #statTonTime[104].Q AND NOT #statPulse[104];   // rising edge
   #statPulse[104] := #statTonTime[104].Q;
   #_w7 := "Unit1.Em8.ControlNodes".hipotThickness.jobInterface.unloadJob4.workingDone OR #_w5 OR ("Unit1.EmNodes".unitStatus.specialFunctions."Dry Run" AND #statUnitStatus.state.idle) OR #_w6;
   IF #_w7 THEN
       "Unit1.Em8.ControlNodes".hipotThickness.jobInterface.loadJob2.workingDone := FALSE;
       "Unit1.Em8.ControlNodes".hipotThickness.jobInterface.inspectionJob3.workingDone := FALSE;
   END_IF;
   IF #_w7 AND FALSE THEN #statPartData := #statDataDelete; END_IF;
END_REGION

REGION Network 28: [Job] Hipot & Thicnkess Guage R*R Select Job
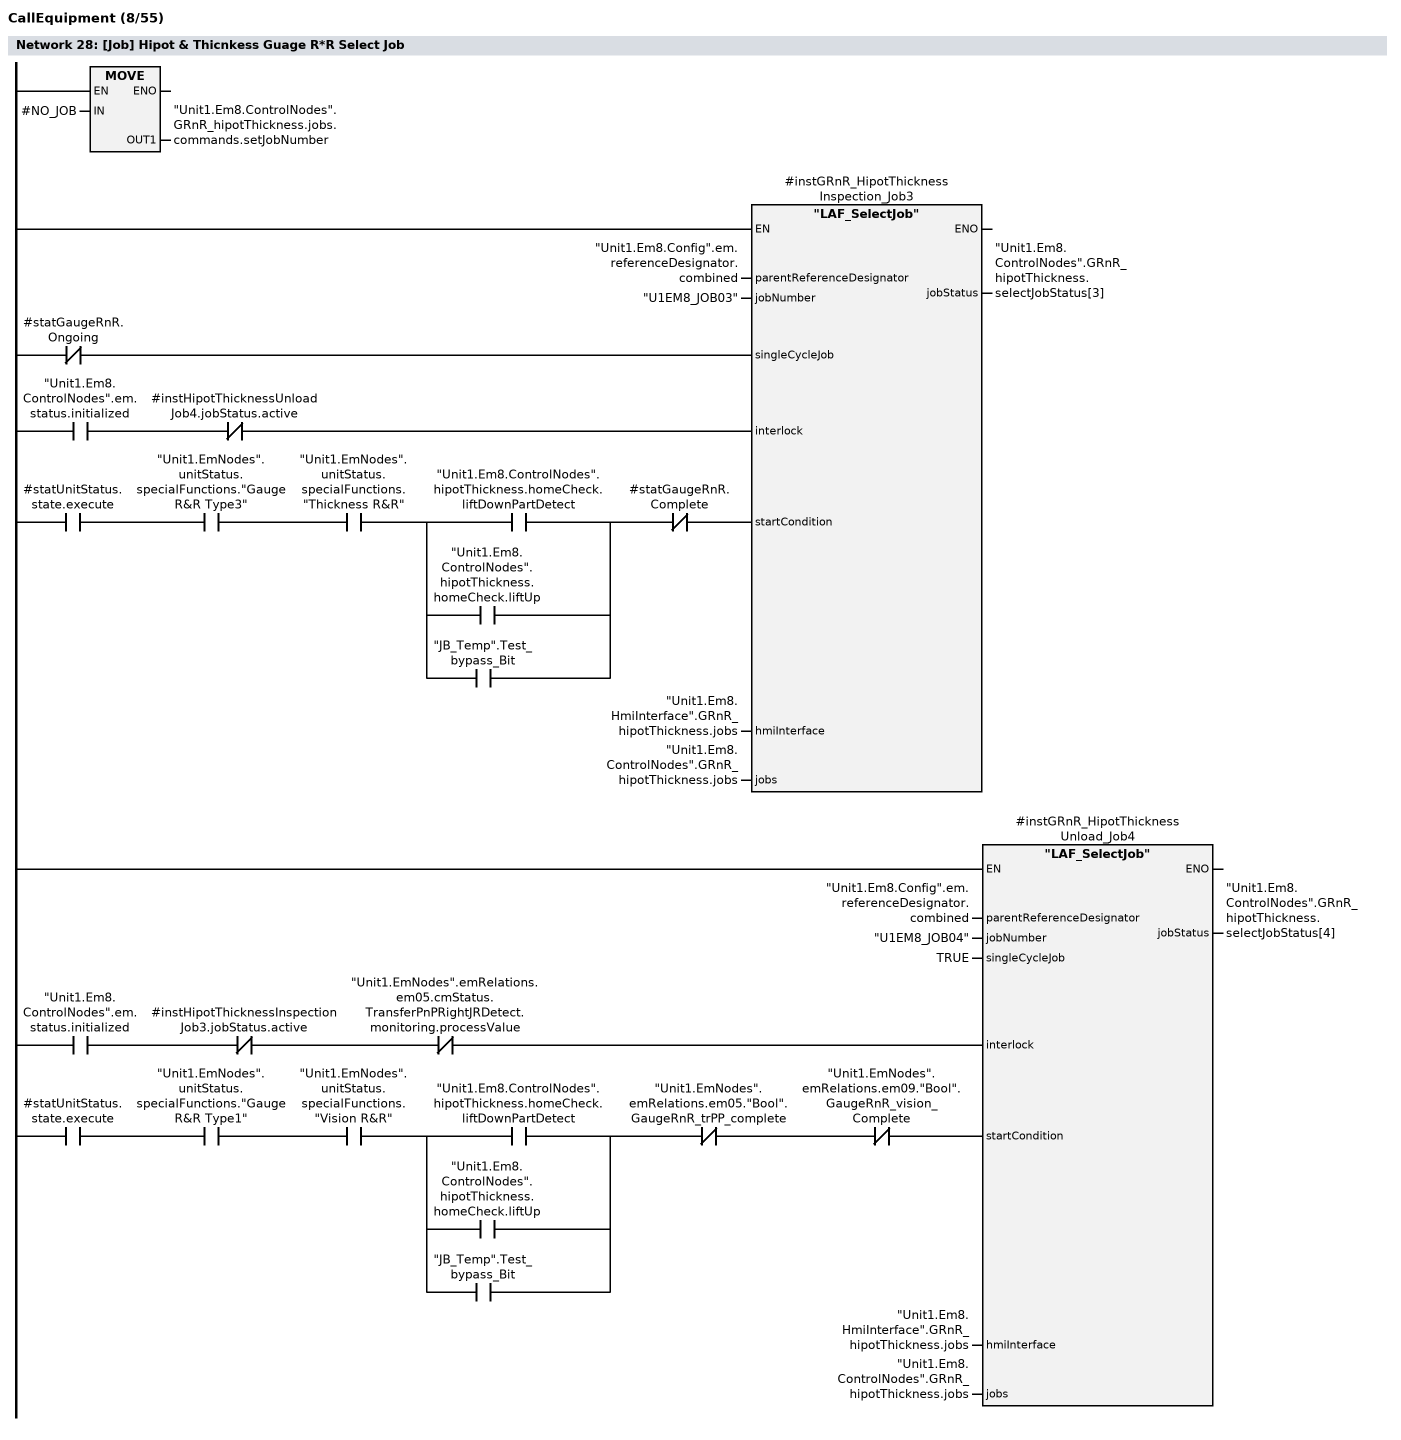
   RUNG wire#powerrail
      Move(in := #NO_JOB, out1 => "Unit1.Em8.ControlNodes".GRnR_hipotThickness.jobs.commands.setJobNumber)
   END_RUNG
   RUNG wire#powerrail
      #instGRnR_HipotThicknessInspection_Job3(singleCycleJob := wire#w1, interlock := wire#w2, startCondition := wire#w5, parentReferenceDesignator := "Unit1.Em8.Config".em.referenceDesignator.combined, jobNumber := "U1EM8_JOB03", hmiInterface := "Unit1.Em8.HmiInterface".GRnR_hipotThickness.jobs, jobs := "Unit1.Em8.ControlNodes".GRnR_hipotThickness.jobs, jobStatus => "Unit1.Em8.ControlNodes".GRnR_hipotThickness.selectJobStatus[3])
   END_RUNG
   RUNG wire#powerrail
      I_Contact( #statGaugeRnR.Ongoing )
   END_RUNG wire#w1
   RUNG wire#powerrail
      Contact( "Unit1.Em8.ControlNodes".em.status.initialized )
      I_Contact( #instHipotThicknessUnloadJob4.jobStatus.active )
   END_RUNG wire#w2
   RUNG wire#powerrail
      Contact( #statUnitStatus.state.execute )
      Contact( "Unit1.EmNodes".unitStatus.specialFunctions."Gauge R&R Type3" )
      Contact( "Unit1.EmNodes".unitStatus.specialFunctions."Thickness R&R" )
      wire#w3
      Contact( "Unit1.Em8.ControlNodes".hipotThickness.homeCheck.liftDownPartDetect )
      wire#w4
      I_Contact( #statGaugeRnR.Complete )
   END_RUNG wire#w5
   RUNG wire#w3
      Contact( "Unit1.Em8.ControlNodes".hipotThickness.homeCheck.liftUp )
   END_RUNG wire#w4
   RUNG wire#w3
      Contact( "JB_Temp".Test_bypass_Bit )
   END_RUNG wire#w4
   RUNG wire#powerrail
      #instGRnR_HipotThicknessUnload_Job4(interlock := wire#w6, startCondition := wire#w9, parentReferenceDesignator := "Unit1.Em8.Config".em.referenceDesignator.combined, jobNumber := "U1EM8_JOB04", singleCycleJob := TRUE, hmiInterface := "Unit1.Em8.HmiInterface".GRnR_hipotThickness.jobs, jobs := "Unit1.Em8.ControlNodes".GRnR_hipotThickness.jobs, jobStatus => "Unit1.Em8.ControlNodes".GRnR_hipotThickness.selectJobStatus[4])
   END_RUNG
   RUNG wire#powerrail
      Contact( "Unit1.Em8.ControlNodes".em.status.initialized )
      I_Contact( #instHipotThicknessInspectionJob3.jobStatus.active )
      I_Contact( "Unit1.EmNodes".emRelations.em05.cmStatus.TransferPnPRightJRDetect.monitoring.processValue )
   END_RUNG wire#w6
   RUNG wire#powerrail
      Contact( #statUnitStatus.state.execute )
      Contact( "Unit1.EmNodes".unitStatus.specialFunctions."Gauge R&R Type1" )
      Contact( "Unit1.EmNodes".unitStatus.specialFunctions."Vision R&R" )
      wire#w7
      Contact( "Unit1.Em8.ControlNodes".hipotThickness.homeCheck.liftDownPartDetect )
      wire#w8
      I_Contact( "Unit1.EmNodes".emRelations.em05."Bool".GaugeRnR_trPP_complete )
      I_Contact( "Unit1.EmNodes".emRelations.em09."Bool".GaugeRnR_vision_Complete )
   END_RUNG wire#w9
   RUNG wire#w7
      Contact( "Unit1.Em8.ControlNodes".hipotThickness.homeCheck.liftUp )
   END_RUNG wire#w8
   RUNG wire#w7
      Contact( "JB_Temp".Test_bypass_Bit )
   END_RUNG wire#w8
   // the same network as SCL:
   "Unit1.Em8.ControlNodes".GRnR_hipotThickness.jobs.commands.setJobNumber := #NO_JOB;
   #instGRnR_HipotThicknessInspection_Job3(parentReferenceDesignator := "Unit1.Em8.Config".em.referenceDesignator.combined,   // "LAF_SelectJob"
                           jobNumber := "U1EM8_JOB03",
                           singleCycleJob := NOT #statGaugeRnR.Ongoing,
                           interlock := "Unit1.Em8.ControlNodes".em.status.initialized AND NOT #instHipotThicknessUnloadJob4.jobStatus.active,
                           startCondition := #statUnitStatus.state.execute AND "Unit1.EmNodes".unitStatus.specialFunctions."Gauge R&R Type3" AND "Unit1.EmNodes".unitStatus.specialFunctions."Thickness R&R" AND ("Unit1.Em8.ControlNodes".hipotThickness.homeCheck.liftDownPartDetect OR "Unit1.Em8.ControlNodes".hipotThickness.homeCheck.liftUp OR "JB_Temp".Test_bypass_Bit) AND NOT #statGaugeRnR.Complete,
                           hmiInterface := "Unit1.Em8.HmiInterface".GRnR_hipotThickness.jobs,
                           jobs := "Unit1.Em8.ControlNodes".GRnR_hipotThickness.jobs,
                           jobStatus => "Unit1.Em8.ControlNodes".GRnR_hipotThickness.selectJobStatus[3]);
   #instGRnR_HipotThicknessUnload_Job4(parentReferenceDesignator := "Unit1.Em8.Config".em.referenceDesignator.combined,   // "LAF_SelectJob"
                           jobNumber := "U1EM8_JOB04",
                           singleCycleJob := TRUE,
                           interlock := "Unit1.Em8.ControlNodes".em.status.initialized AND NOT #instHipotThicknessInspectionJob3.jobStatus.active AND NOT "Unit1.EmNodes".emRelations.em05.cmStatus.TransferPnPRightJRDetect.monitoring.processValue,
                           startCondition := #statUnitStatus.state.execute AND "Unit1.EmNodes".unitStatus.specialFunctions."Gauge R&R Type1" AND "Unit1.EmNodes".unitStatus.specialFunctions."Vision R&R" AND ("Unit1.Em8.ControlNodes".hipotThickness.homeCheck.liftDownPartDetect OR "Unit1.Em8.ControlNodes".hipotThickness.homeCheck.liftUp OR "JB_Temp".Test_bypass_Bit) AND NOT "Unit1.EmNodes".emRelations.em05."Bool".GaugeRnR_trPP_complete AND NOT "Unit1.EmNodes".emRelations.em09."Bool".GaugeRnR_vision_Complete,
                           hmiInterface := "Unit1.Em8.HmiInterface".GRnR_hipotThickness.jobs,
                           jobs := "Unit1.Em8.ControlNodes".GRnR_hipotThickness.jobs,
                           jobStatus => "Unit1.Em8.ControlNodes".GRnR_hipotThickness.selectJobStatus[4]);
END_REGION

REGION Network 29: Guage RnR Hipot & Thickness Job Interface [Unloading]
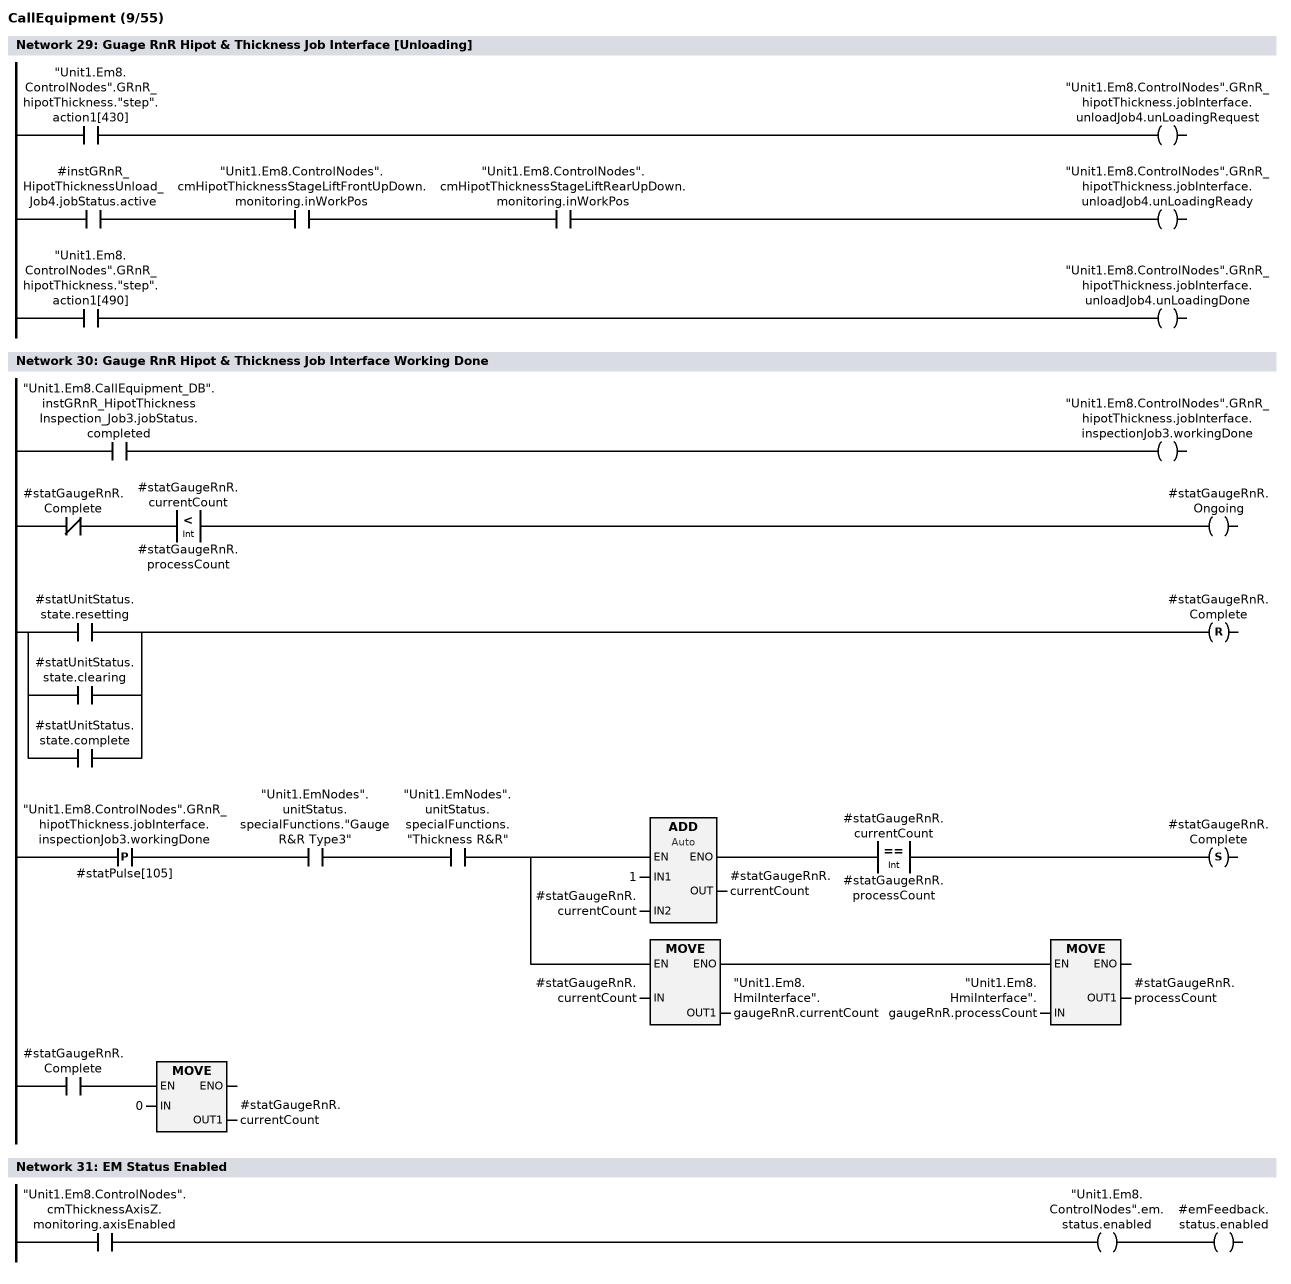
   RUNG wire#powerrail
      Contact( "Unit1.Em8.ControlNodes".GRnR_hipotThickness."step".action1[430] )
      Coil( "Unit1.Em8.ControlNodes".GRnR_hipotThickness.jobInterface.unloadJob4.unLoadingRequest )
   END_RUNG
   RUNG wire#powerrail
      Contact( #instGRnR_HipotThicknessUnload_Job4.jobStatus.active )
      Contact( "Unit1.Em8.ControlNodes".cmHipotThicknessStageLiftFrontUpDown.monitoring.inWorkPos )
      Contact( "Unit1.Em8.ControlNodes".cmHipotThicknessStageLiftRearUpDown.monitoring.inWorkPos )
      Coil( "Unit1.Em8.ControlNodes".GRnR_hipotThickness.jobInterface.unloadJob4.unLoadingReady )
   END_RUNG
   RUNG wire#powerrail
      Contact( "Unit1.Em8.ControlNodes".GRnR_hipotThickness."step".action1[490] )
      Coil( "Unit1.Em8.ControlNodes".GRnR_hipotThickness.jobInterface.unloadJob4.unLoadingDone )
   END_RUNG
   // the same network as SCL:
   "Unit1.Em8.ControlNodes".GRnR_hipotThickness.jobInterface.unloadJob4.unLoadingRequest := "Unit1.Em8.ControlNodes".GRnR_hipotThickness."step".action1[430];
   "Unit1.Em8.ControlNodes".GRnR_hipotThickness.jobInterface.unloadJob4.unLoadingReady := #instGRnR_HipotThicknessUnload_Job4.jobStatus.active AND "Unit1.Em8.ControlNodes".cmHipotThicknessStageLiftFrontUpDown.monitoring.inWorkPos AND "Unit1.Em8.ControlNodes".cmHipotThicknessStageLiftRearUpDown.monitoring.inWorkPos;
   "Unit1.Em8.ControlNodes".GRnR_hipotThickness.jobInterface.unloadJob4.unLoadingDone := "Unit1.Em8.ControlNodes".GRnR_hipotThickness."step".action1[490];
END_REGION

REGION Network 30: Gauge RnR Hipot & Thickness Job Interface Working Done
   RUNG wire#powerrail
      Contact( "Unit1.Em8.CallEquipment_DB".instGRnR_HipotThicknessInspection_Job3.jobStatus.completed )
      Coil( "Unit1.Em8.ControlNodes".GRnR_hipotThickness.jobInterface.inspectionJob3.workingDone )
   END_RUNG
   RUNG wire#powerrail
      I_Contact( #statGaugeRnR.Complete )
      { S7_Templates := "SrcType := Int" } LT_Contact(in1 := #statGaugeRnR.currentCount, in2 := #statGaugeRnR.processCount)
      Coil( #statGaugeRnR.Ongoing )
   END_RUNG
   RUNG wire#powerrail
      Contact( #statUnitStatus.state.resetting )
      wire#w1
      R_Coil( #statGaugeRnR.Complete )
   END_RUNG
   RUNG wire#powerrail
      Contact( #statUnitStatus.state.clearing )
   END_RUNG wire#w1
   RUNG wire#powerrail
      Contact( #statUnitStatus.state.complete )
   END_RUNG wire#w1
   RUNG wire#powerrail
      P_Contact(operand := "Unit1.Em8.ControlNodes".GRnR_hipotThickness.jobInterface.inspectionJob3.workingDone, bit := #statPulse[105])
      Contact( "Unit1.EmNodes".unitStatus.specialFunctions."Gauge R&R Type3" )
      Contact( "Unit1.EmNodes".unitStatus.specialFunctions."Thickness R&R" )
      wire#w2
      Add(in1 := 1, in2 := #statGaugeRnR.currentCount, out => #statGaugeRnR.currentCount)
      { S7_Templates := "SrcType := Int" } EQ_Contact(in1 := #statGaugeRnR.currentCount, in2 := #statGaugeRnR.processCount)
      S_Coil( #statGaugeRnR.Complete )
   END_RUNG
   RUNG wire#w2
      Move(in := #statGaugeRnR.currentCount, out1 => "Unit1.Em8.HmiInterface".gaugeRnR.currentCount)
      Move(in := "Unit1.Em8.HmiInterface".gaugeRnR.processCount, out1 => #statGaugeRnR.processCount)
   END_RUNG
   RUNG wire#powerrail
      Contact( #statGaugeRnR.Complete )
      Move(in := 0, out1 => #statGaugeRnR.currentCount)
   END_RUNG
   // the same network as SCL:
   "Unit1.Em8.ControlNodes".GRnR_hipotThickness.jobInterface.inspectionJob3.workingDone := "Unit1.Em8.CallEquipment_DB".instGRnR_HipotThicknessInspection_Job3.jobStatus.completed;
   #statGaugeRnR.Ongoing := NOT #statGaugeRnR.Complete AND (#statGaugeRnR.currentCount < #statGaugeRnR.processCount);
   IF #statUnitStatus.state.resetting OR #statUnitStatus.state.clearing OR #statUnitStatus.state.complete THEN
       #statGaugeRnR.Complete := FALSE;
   END_IF;
   #_w1 := "Unit1.Em8.ControlNodes".GRnR_hipotThickness.jobInterface.inspectionJob3.workingDone AND NOT #statPulse[105];   // rising edge of "Unit1.Em8.ControlNodes".GRnR_hipotThickness.jobInterface.inspectionJob3.workingDone
   #statPulse[105] := "Unit1.Em8.ControlNodes".GRnR_hipotThickness.jobInterface.inspectionJob3.workingDone;
   #_w2 := #_w1 AND "Unit1.EmNodes".unitStatus.specialFunctions."Gauge R&R Type3" AND "Unit1.EmNodes".unitStatus.specialFunctions."Thickness R&R";
   IF #_w2 THEN #statGaugeRnR.currentCount := 1 + #statGaugeRnR.currentCount; END_IF;
   IF #_w2 AND (#statGaugeRnR.currentCount = #statGaugeRnR.processCount) THEN
       #statGaugeRnR.Complete := TRUE;
   END_IF;
   IF #_w2 THEN
       "Unit1.Em8.HmiInterface".gaugeRnR.currentCount := #statGaugeRnR.currentCount;
       #statGaugeRnR.processCount := "Unit1.Em8.HmiInterface".gaugeRnR.processCount;
   END_IF;
   IF #statGaugeRnR.Complete THEN #statGaugeRnR.currentCount := 0; END_IF;
END_REGION

REGION Network 31: EM Status Enabled
   RUNG wire#powerrail
      Contact( "Unit1.Em8.ControlNodes".cmThicknessAxisZ.monitoring.axisEnabled )
      Coil( "Unit1.Em8.ControlNodes".em.status.enabled )
      Coil( #emFeedback.status.enabled )
   END_RUNG
   // the same network as SCL:
   "Unit1.Em8.ControlNodes".em.status.enabled := "Unit1.Em8.ControlNodes".cmThicknessAxisZ.monitoring.axisEnabled;
   #emFeedback.status.enabled := "Unit1.Em8.ControlNodes".cmThicknessAxisZ.monitoring.axisEnabled;
END_REGION

REGION Network 32: Set EM To Initialized
   // Set em to initialized here. Usually this is done when the initialization job is completed.
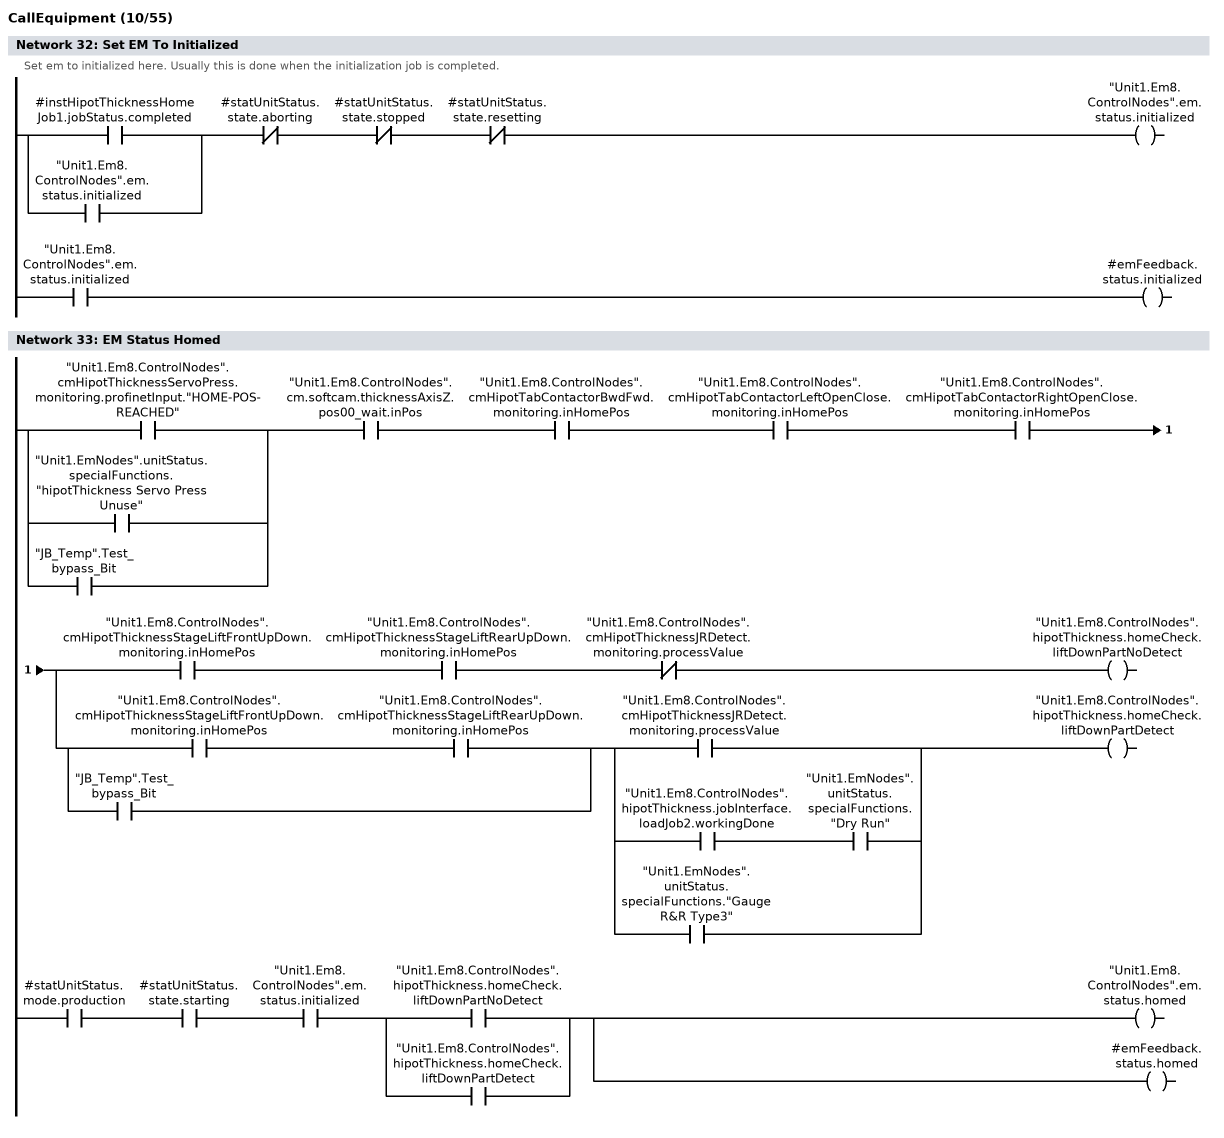
   RUNG wire#powerrail
      Contact( #instHipotThicknessHomeJob1.jobStatus.completed )
      wire#w1
      I_Contact( #statUnitStatus.state.aborting )
      I_Contact( #statUnitStatus.state.stopped )
      I_Contact( #statUnitStatus.state.resetting )
      Coil( "Unit1.Em8.ControlNodes".em.status.initialized )
   END_RUNG
   RUNG wire#powerrail
      Contact( "Unit1.Em8.ControlNodes".em.status.initialized )
   END_RUNG wire#w1
   RUNG wire#powerrail
      Contact( "Unit1.Em8.ControlNodes".em.status.initialized )
      Coil( #emFeedback.status.initialized )
   END_RUNG
   // the same network as SCL:
   "Unit1.Em8.ControlNodes".em.status.initialized := (#instHipotThicknessHomeJob1.jobStatus.completed OR "Unit1.Em8.ControlNodes".em.status.initialized) AND NOT #statUnitStatus.state.aborting AND NOT #statUnitStatus.state.stopped AND NOT #statUnitStatus.state.resetting;
   #emFeedback.status.initialized := "Unit1.Em8.ControlNodes".em.status.initialized;
END_REGION

REGION Network 33: EM Status Homed
   RUNG wire#powerrail
      Contact( "Unit1.Em8.ControlNodes".cmHipotThicknessServoPress.monitoring.profinetInput."HOME-POS-REACHED" )
      wire#w1
      Contact( "Unit1.Em8.ControlNodes".cm.softcam.thicknessAxisZ.pos00_wait.inPos )
      Contact( "Unit1.Em8.ControlNodes".cmHipotTabContactorBwdFwd.monitoring.inHomePos )
      Contact( "Unit1.Em8.ControlNodes".cmHipotTabContactorLeftOpenClose.monitoring.inHomePos )
      Contact( "Unit1.Em8.ControlNodes".cmHipotTabContactorRightOpenClose.monitoring.inHomePos )
      wire#w2
      Contact( "Unit1.Em8.ControlNodes".cmHipotThicknessStageLiftFrontUpDown.monitoring.inHomePos )
      Contact( "Unit1.Em8.ControlNodes".cmHipotThicknessStageLiftRearUpDown.monitoring.inHomePos )
      I_Contact( "Unit1.Em8.ControlNodes".cmHipotThicknessJRDetect.monitoring.processValue )
      Coil( "Unit1.Em8.ControlNodes".hipotThickness.homeCheck.liftDownPartNoDetect )
   END_RUNG
   RUNG wire#powerrail
      Contact( "Unit1.EmNodes".unitStatus.specialFunctions."hipotThickness Servo Press Unuse" )
   END_RUNG wire#w1
   RUNG wire#powerrail
      Contact( "JB_Temp".Test_bypass_Bit )
   END_RUNG wire#w1
   RUNG wire#w2
      Contact( "Unit1.Em8.ControlNodes".cmHipotThicknessStageLiftFrontUpDown.monitoring.inHomePos )
      Contact( "Unit1.Em8.ControlNodes".cmHipotThicknessStageLiftRearUpDown.monitoring.inHomePos )
      wire#w3
      Contact( "Unit1.Em8.ControlNodes".cmHipotThicknessJRDetect.monitoring.processValue )
      wire#w4
      Coil( "Unit1.Em8.ControlNodes".hipotThickness.homeCheck.liftDownPartDetect )
   END_RUNG
   RUNG wire#w2
      Contact( "JB_Temp".Test_bypass_Bit )
   END_RUNG wire#w3
   RUNG wire#w3
      Contact( "Unit1.Em8.ControlNodes".hipotThickness.jobInterface.loadJob2.workingDone )
      Contact( "Unit1.EmNodes".unitStatus.specialFunctions."Dry Run" )
   END_RUNG wire#w4
   RUNG wire#w3
      Contact( "Unit1.EmNodes".unitStatus.specialFunctions."Gauge R&R Type3" )
   END_RUNG wire#w4
   RUNG wire#powerrail
      Contact( #statUnitStatus.mode.production )
      Contact( #statUnitStatus.state.starting )
      Contact( "Unit1.Em8.ControlNodes".em.status.initialized )
      wire#w5
      Contact( "Unit1.Em8.ControlNodes".hipotThickness.homeCheck.liftDownPartNoDetect )
      wire#w6
      Coil( "Unit1.Em8.ControlNodes".em.status.homed )
   END_RUNG
   RUNG wire#w5
      Contact( "Unit1.Em8.ControlNodes".hipotThickness.homeCheck.liftDownPartDetect )
   END_RUNG wire#w6
   RUNG wire#w6
      Coil( #emFeedback.status.homed )
   END_RUNG
   // the same network as SCL:
   #_w1 := ("Unit1.Em8.ControlNodes".cmHipotThicknessServoPress.monitoring.profinetInput."HOME-POS-REACHED" OR "Unit1.EmNodes".unitStatus.specialFunctions."hipotThickness Servo Press Unuse" OR "JB_Temp".Test_bypass_Bit) AND "Unit1.Em8.ControlNodes".cm.softcam.thicknessAxisZ.pos00_wait.inPos AND "Unit1.Em8.ControlNodes".cmHipotTabContactorBwdFwd.monitoring.inHomePos AND "Unit1.Em8.ControlNodes".cmHipotTabContactorLeftOpenClose.monitoring.inHomePos AND "Unit1.Em8.ControlNodes".cmHipotTabContactorRightOpenClose.monitoring.inHomePos;
   "Unit1.Em8.ControlNodes".hipotThickness.homeCheck.liftDownPartNoDetect := #_w1 AND "Unit1.Em8.ControlNodes".cmHipotThicknessStageLiftFrontUpDown.monitoring.inHomePos AND "Unit1.Em8.ControlNodes".cmHipotThicknessStageLiftRearUpDown.monitoring.inHomePos AND NOT "Unit1.Em8.ControlNodes".cmHipotThicknessJRDetect.monitoring.processValue;
   "Unit1.Em8.ControlNodes".hipotThickness.homeCheck.liftDownPartDetect := #_w1 AND (("Unit1.Em8.ControlNodes".cmHipotThicknessStageLiftFrontUpDown.monitoring.inHomePos AND "Unit1.Em8.ControlNodes".cmHipotThicknessStageLiftRearUpDown.monitoring.inHomePos) OR "JB_Temp".Test_bypass_Bit) AND ("Unit1.Em8.ControlNodes".cmHipotThicknessJRDetect.monitoring.processValue OR ("Unit1.Em8.ControlNodes".hipotThickness.jobInterface.loadJob2.workingDone AND "Unit1.EmNodes".unitStatus.specialFunctions."Dry Run") OR "Unit1.EmNodes".unitStatus.specialFunctions."Gauge R&R Type3");
   "Unit1.Em8.ControlNodes".em.status.homed := #statUnitStatus.mode.production AND #statUnitStatus.state.starting AND "Unit1.Em8.ControlNodes".em.status.initialized AND ("Unit1.Em8.ControlNodes".hipotThickness.homeCheck.liftDownPartNoDetect OR "Unit1.Em8.ControlNodes".hipotThickness.homeCheck.liftDownPartDetect);
   #emFeedback.status.homed := "Unit1.Em8.ControlNodes".em.status.homed;
END_REGION

REGION Network 34: Position Check
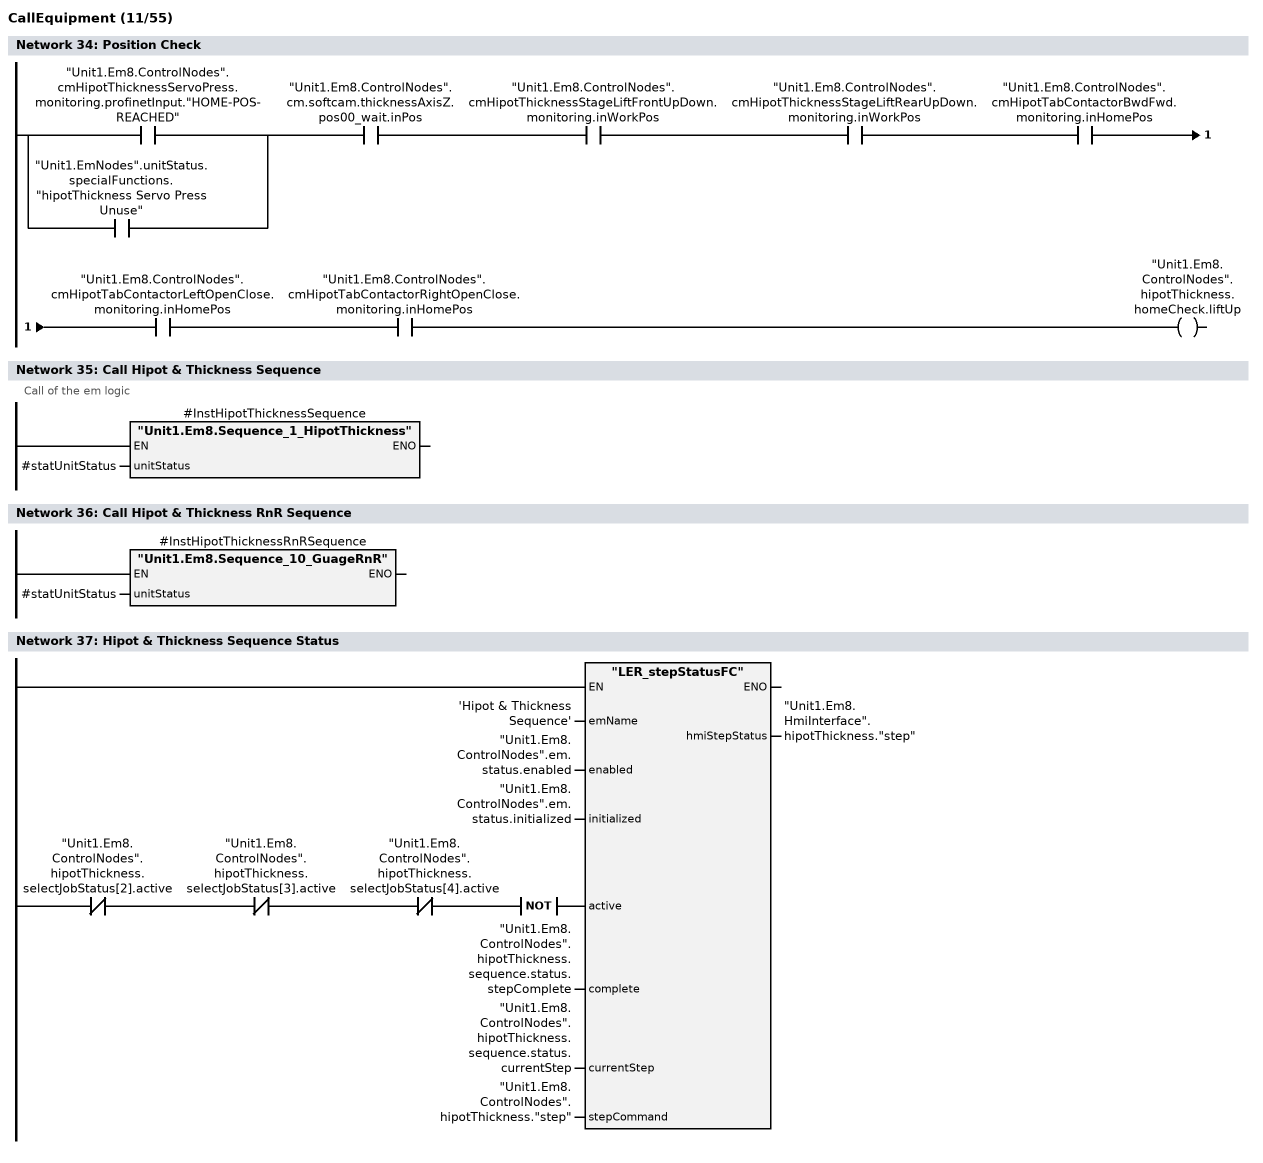
   RUNG wire#powerrail
      Contact( "Unit1.Em8.ControlNodes".cmHipotThicknessServoPress.monitoring.profinetInput."HOME-POS-REACHED" )
      wire#w1
      Contact( "Unit1.Em8.ControlNodes".cm.softcam.thicknessAxisZ.pos00_wait.inPos )
      Contact( "Unit1.Em8.ControlNodes".cmHipotThicknessStageLiftFrontUpDown.monitoring.inWorkPos )
      Contact( "Unit1.Em8.ControlNodes".cmHipotThicknessStageLiftRearUpDown.monitoring.inWorkPos )
      Contact( "Unit1.Em8.ControlNodes".cmHipotTabContactorBwdFwd.monitoring.inHomePos )
      Contact( "Unit1.Em8.ControlNodes".cmHipotTabContactorLeftOpenClose.monitoring.inHomePos )
      Contact( "Unit1.Em8.ControlNodes".cmHipotTabContactorRightOpenClose.monitoring.inHomePos )
      Coil( "Unit1.Em8.ControlNodes".hipotThickness.homeCheck.liftUp )
   END_RUNG
   RUNG wire#powerrail
      Contact( "Unit1.EmNodes".unitStatus.specialFunctions."hipotThickness Servo Press Unuse" )
   END_RUNG wire#w1
   // the same network as SCL:
   "Unit1.Em8.ControlNodes".hipotThickness.homeCheck.liftUp := ("Unit1.Em8.ControlNodes".cmHipotThicknessServoPress.monitoring.profinetInput."HOME-POS-REACHED" OR "Unit1.EmNodes".unitStatus.specialFunctions."hipotThickness Servo Press Unuse") AND "Unit1.Em8.ControlNodes".cm.softcam.thicknessAxisZ.pos00_wait.inPos AND "Unit1.Em8.ControlNodes".cmHipotThicknessStageLiftFrontUpDown.monitoring.inWorkPos AND "Unit1.Em8.ControlNodes".cmHipotThicknessStageLiftRearUpDown.monitoring.inWorkPos AND "Unit1.Em8.ControlNodes".cmHipotTabContactorBwdFwd.monitoring.inHomePos AND "Unit1.Em8.ControlNodes".cmHipotTabContactorLeftOpenClose.monitoring.inHomePos AND "Unit1.Em8.ControlNodes".cmHipotTabContactorRightOpenClose.monitoring.inHomePos;
END_REGION

REGION Network 35: Call Hipot & Thickness Sequence
   // Call of the em logic
   RUNG wire#powerrail
      #InstHipotThicknessSequence(unitStatus := #statUnitStatus)
   END_RUNG
   // the same network as SCL:
   #InstHipotThicknessSequence(unitStatus := #statUnitStatus);   // "Unit1.Em8.Sequence_1_HipotThickness"
END_REGION

REGION Network 36: Call Hipot & Thickness RnR Sequence
   RUNG wire#powerrail
      #InstHipotThicknessRnRSequence(unitStatus := #statUnitStatus)
   END_RUNG
   // the same network as SCL:
   #InstHipotThicknessRnRSequence(unitStatus := #statUnitStatus);   // "Unit1.Em8.Sequence_10_GuageRnR"
END_REGION

REGION Network 37: Hipot & Thickness Sequence Status
   RUNG wire#powerrail
      "LER_stepStatusFC"(active := wire#w1, emName := 'Hipot & Thickness Sequence', enabled := "Unit1.Em8.ControlNodes".em.status.enabled, initialized := "Unit1.Em8.ControlNodes".em.status.initialized, complete := "Unit1.Em8.ControlNodes".hipotThickness.sequence.status.stepComplete, currentStep := "Unit1.Em8.ControlNodes".hipotThickness.sequence.status.currentStep, stepCommand := "Unit1.Em8.ControlNodes".hipotThickness."step", hmiStepStatus => "Unit1.Em8.HmiInterface".hipotThickness."step")
   END_RUNG
   RUNG wire#powerrail
      I_Contact( "Unit1.Em8.ControlNodes".hipotThickness.selectJobStatus[2].active )
      I_Contact( "Unit1.Em8.ControlNodes".hipotThickness.selectJobStatus[3].active )
      I_Contact( "Unit1.Em8.ControlNodes".hipotThickness.selectJobStatus[4].active )
      Not()
   END_RUNG wire#w1
   // the same network as SCL:
   "LER_stepStatusFC"(emName := 'Hipot & Thickness Sequence',
                      enabled := "Unit1.Em8.ControlNodes".em.status.enabled,
                      initialized := "Unit1.Em8.ControlNodes".em.status.initialized,
                      active := NOT (NOT "Unit1.Em8.ControlNodes".hipotThickness.selectJobStatus[2].active AND NOT "Unit1.Em8.ControlNodes".hipotThickness.selectJobStatus[3].active AND NOT "Unit1.Em8.ControlNodes".hipotThickness.selectJobStatus[4].active),
                      complete := "Unit1.Em8.ControlNodes".hipotThickness.sequence.status.stepComplete,
                      currentStep := "Unit1.Em8.ControlNodes".hipotThickness.sequence.status.currentStep,
                      stepCommand := "Unit1.Em8.ControlNodes".hipotThickness."step",
                      hmiStepStatus => "Unit1.Em8.HmiInterface".hipotThickness."step");
END_REGION

REGION Network 38: Hipot & Thickness RnR Sequence Status
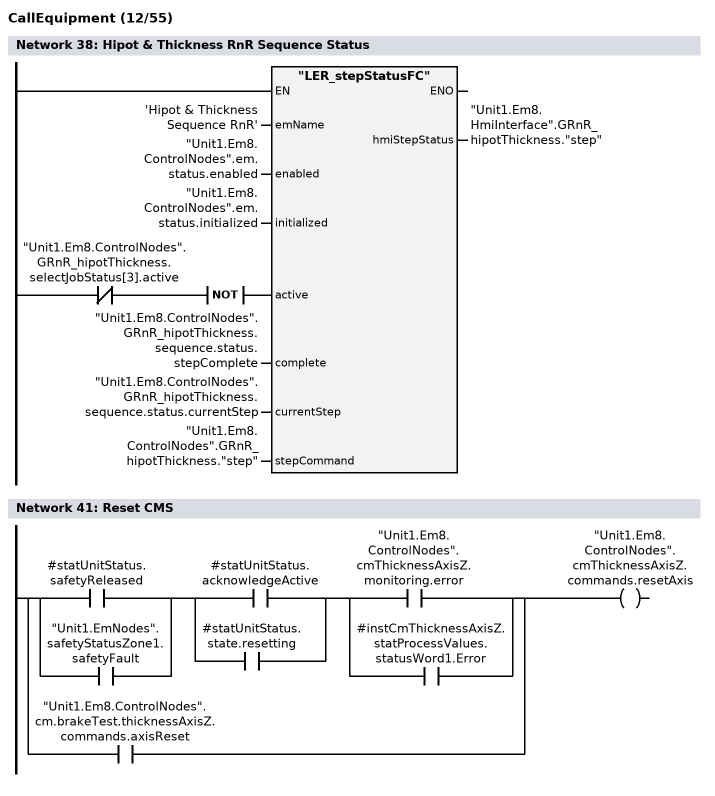
   RUNG wire#powerrail
      "LER_stepStatusFC"(active := wire#w1, emName := 'Hipot & Thickness Sequence RnR', enabled := "Unit1.Em8.ControlNodes".em.status.enabled, initialized := "Unit1.Em8.ControlNodes".em.status.initialized, complete := "Unit1.Em8.ControlNodes".GRnR_hipotThickness.sequence.status.stepComplete, currentStep := "Unit1.Em8.ControlNodes".GRnR_hipotThickness.sequence.status.currentStep, stepCommand := "Unit1.Em8.ControlNodes".GRnR_hipotThickness."step", hmiStepStatus => "Unit1.Em8.HmiInterface".GRnR_hipotThickness."step")
   END_RUNG
   RUNG wire#powerrail
      I_Contact( "Unit1.Em8.ControlNodes".GRnR_hipotThickness.selectJobStatus[3].active )
      Not()
   END_RUNG wire#w1
   // the same network as SCL:
   "LER_stepStatusFC"(emName := 'Hipot & Thickness Sequence RnR',
                      enabled := "Unit1.Em8.ControlNodes".em.status.enabled,
                      initialized := "Unit1.Em8.ControlNodes".em.status.initialized,
                      active := NOT (NOT "Unit1.Em8.ControlNodes".GRnR_hipotThickness.selectJobStatus[3].active),
                      complete := "Unit1.Em8.ControlNodes".GRnR_hipotThickness.sequence.status.stepComplete,
                      currentStep := "Unit1.Em8.ControlNodes".GRnR_hipotThickness.sequence.status.currentStep,
                      stepCommand := "Unit1.Em8.ControlNodes".GRnR_hipotThickness."step",
                      hmiStepStatus => "Unit1.Em8.HmiInterface".GRnR_hipotThickness."step");
END_REGION

REGION Network 40: ******************** Control Modules (Axis) ********************
   // Call control modules that are sensors before the em logic (jobs and sequence), so that the latest value is used in the logic.
END_REGION

REGION Network 41: Reset CMS
   RUNG wire#powerrail
      Contact( #statUnitStatus.safetyReleased )
      wire#w1
      Contact( #statUnitStatus.acknowledgeActive )
      wire#w2
      Contact( "Unit1.Em8.ControlNodes".cmThicknessAxisZ.monitoring.error )
      wire#w3
      Coil( "Unit1.Em8.ControlNodes".cmThicknessAxisZ.commands.resetAxis )
   END_RUNG
   RUNG wire#powerrail
      Contact( "Unit1.EmNodes".safetyStatusZone1.safetyFault )
   END_RUNG wire#w1
   RUNG wire#w1
      Contact( #statUnitStatus.state.resetting )
   END_RUNG wire#w2
   RUNG wire#w2
      Contact( #instCmThicknessAxisZ.statProcessValues.statusWord1.Error )
   END_RUNG wire#w3
   RUNG wire#powerrail
      Contact( "Unit1.Em8.ControlNodes".cm.brakeTest.thicknessAxisZ.commands.axisReset )
   END_RUNG wire#w3
   // the same network as SCL:
   "Unit1.Em8.ControlNodes".cmThicknessAxisZ.commands.resetAxis := ((#statUnitStatus.safetyReleased OR "Unit1.EmNodes".safetyStatusZone1.safetyFault) AND (#statUnitStatus.acknowledgeActive OR #statUnitStatus.state.resetting) AND ("Unit1.Em8.ControlNodes".cmThicknessAxisZ.monitoring.error OR #instCmThicknessAxisZ.statProcessValues.statusWord1.Error)) OR "Unit1.Em8.ControlNodes".cm.brakeTest.thicknessAxisZ.commands.axisReset;
END_REGION

REGION Network 42: Enable/Disable CMS
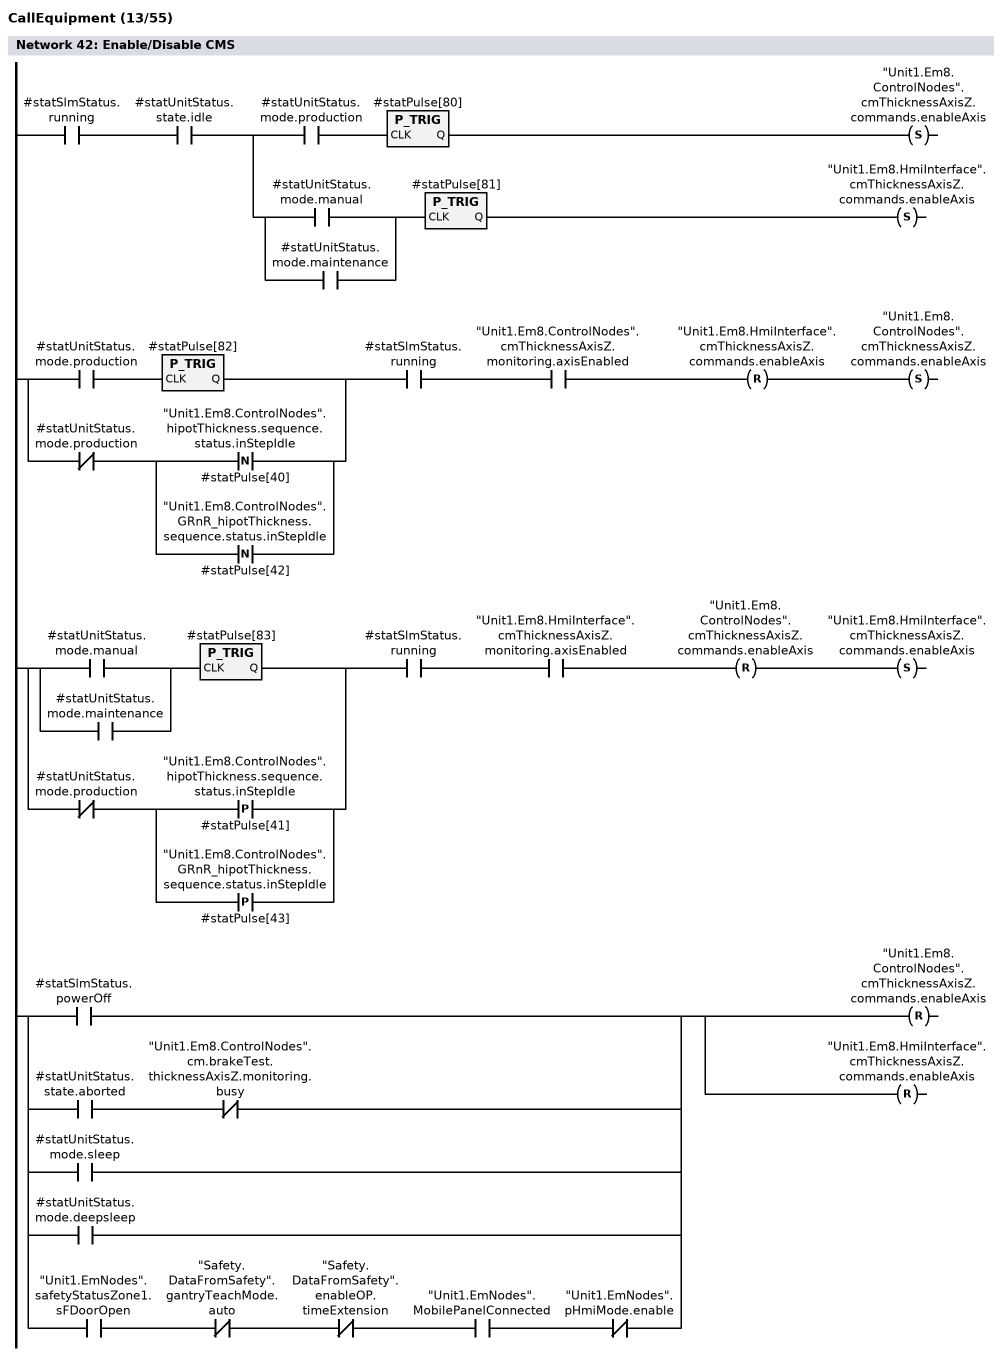
   RUNG wire#powerrail
      Contact( #statSlmStatus.running )
      Contact( #statUnitStatus.state.idle )
      wire#w1
      Contact( #statUnitStatus.mode.production )
      P_Trig( #statPulse[80] )
      S_Coil( "Unit1.Em8.ControlNodes".cmThicknessAxisZ.commands.enableAxis )
   END_RUNG
   RUNG wire#w1
      Contact( #statUnitStatus.mode.manual )
      wire#w2
      P_Trig( #statPulse[81] )
      S_Coil( "Unit1.Em8.HmiInterface".cmThicknessAxisZ.commands.enableAxis )
   END_RUNG
   RUNG wire#w1
      Contact( #statUnitStatus.mode.maintenance )
   END_RUNG wire#w2
   RUNG wire#powerrail
      Contact( #statUnitStatus.mode.production )
      P_Trig( #statPulse[82] )
      wire#w3
      Contact( #statSlmStatus.running )
      Contact( "Unit1.Em8.ControlNodes".cmThicknessAxisZ.monitoring.axisEnabled )
      R_Coil( "Unit1.Em8.HmiInterface".cmThicknessAxisZ.commands.enableAxis )
      S_Coil( "Unit1.Em8.ControlNodes".cmThicknessAxisZ.commands.enableAxis )
   END_RUNG
   RUNG wire#powerrail
      I_Contact( #statUnitStatus.mode.production )
      wire#w4
      N_Contact(operand := "Unit1.Em8.ControlNodes".hipotThickness.sequence.status.inStepIdle, bit := #statPulse[40])
   END_RUNG wire#w3
   RUNG wire#w4
      N_Contact(operand := "Unit1.Em8.ControlNodes".GRnR_hipotThickness.sequence.status.inStepIdle, bit := #statPulse[42])
   END_RUNG wire#w3
   RUNG wire#powerrail
      Contact( #statUnitStatus.mode.manual )
      wire#w5
      P_Trig( #statPulse[83] )
      wire#w6
      Contact( #statSlmStatus.running )
      Contact( "Unit1.Em8.HmiInterface".cmThicknessAxisZ.monitoring.axisEnabled )
      R_Coil( "Unit1.Em8.ControlNodes".cmThicknessAxisZ.commands.enableAxis )
      S_Coil( "Unit1.Em8.HmiInterface".cmThicknessAxisZ.commands.enableAxis )
   END_RUNG
   RUNG wire#powerrail
      Contact( #statUnitStatus.mode.maintenance )
   END_RUNG wire#w5
   RUNG wire#powerrail
      I_Contact( #statUnitStatus.mode.production )
      wire#w7
      P_Contact(operand := "Unit1.Em8.ControlNodes".hipotThickness.sequence.status.inStepIdle, bit := #statPulse[41])
   END_RUNG wire#w6
   RUNG wire#w7
      P_Contact(operand := "Unit1.Em8.ControlNodes".GRnR_hipotThickness.sequence.status.inStepIdle, bit := #statPulse[43])
   END_RUNG wire#w6
   RUNG wire#powerrail
      Contact( #statSlmStatus.powerOff )
      wire#w8
      R_Coil( "Unit1.Em8.ControlNodes".cmThicknessAxisZ.commands.enableAxis )
   END_RUNG
   RUNG wire#powerrail
      Contact( #statUnitStatus.state.aborted )
      I_Contact( "Unit1.Em8.ControlNodes".cm.brakeTest.thicknessAxisZ.monitoring.busy )
   END_RUNG wire#w8
   RUNG wire#powerrail
      Contact( #statUnitStatus.mode.sleep )
   END_RUNG wire#w8
   RUNG wire#powerrail
      Contact( #statUnitStatus.mode.deepsleep )
   END_RUNG wire#w8
   RUNG wire#powerrail
      Contact( "Unit1.EmNodes".safetyStatusZone1.sFDoorOpen )
      I_Contact( "Safety.DataFromSafety".gantryTeachMode.auto )
      I_Contact( "Safety.DataFromSafety".enableOP.timeExtension )
      Contact( "Unit1.EmNodes".MobilePanelConnected )
      I_Contact( "Unit1.EmNodes".pHmiMode.enable )
   END_RUNG wire#w8
   RUNG wire#w8
      R_Coil( "Unit1.Em8.HmiInterface".cmThicknessAxisZ.commands.enableAxis )
   END_RUNG
   // the same network as SCL:
   #_w1 := #statSlmStatus.running AND #statUnitStatus.state.idle;
   #_w2 := #_w1 AND #statUnitStatus.mode.production;
   #_w3 := #_w2 AND NOT #statPulse[80];   // rising edge
   #statPulse[80] := #_w2;
   IF #_w3 THEN "Unit1.Em8.ControlNodes".cmThicknessAxisZ.commands.enableAxis := TRUE; END_IF;
   #_w4 := #_w1 AND (#statUnitStatus.mode.manual OR #statUnitStatus.mode.maintenance);
   #_w5 := #_w4 AND NOT #statPulse[81];   // rising edge
   #statPulse[81] := #_w4;
   IF #_w5 THEN "Unit1.Em8.HmiInterface".cmThicknessAxisZ.commands.enableAxis := TRUE; END_IF;
   #_w6 := #statUnitStatus.mode.production AND NOT #statPulse[82];   // rising edge
   #statPulse[82] := #statUnitStatus.mode.production;
   #_w7 := NOT #statUnitStatus.mode.production AND NOT "Unit1.Em8.ControlNodes".hipotThickness.sequence.status.inStepIdle AND #statPulse[40];   // falling edge of "Unit1.Em8.ControlNodes".hipotThickness.sequence.status.inStepIdle
   #statPulse[40] := "Unit1.Em8.ControlNodes".hipotThickness.sequence.status.inStepIdle;
   #_w8 := NOT #statUnitStatus.mode.production AND NOT "Unit1.Em8.ControlNodes".GRnR_hipotThickness.sequence.status.inStepIdle AND #statPulse[42];   // falling edge of "Unit1.Em8.ControlNodes".GRnR_hipotThickness.sequence.status.inStepIdle
   #statPulse[42] := "Unit1.Em8.ControlNodes".GRnR_hipotThickness.sequence.status.inStepIdle;
   IF (#_w6 OR #_w7 OR #_w8) AND #statSlmStatus.running AND "Unit1.Em8.ControlNodes".cmThicknessAxisZ.monitoring.axisEnabled THEN
       "Unit1.Em8.HmiInterface".cmThicknessAxisZ.commands.enableAxis := FALSE;
       "Unit1.Em8.ControlNodes".cmThicknessAxisZ.commands.enableAxis := TRUE;
   END_IF;
   #_w9 := #statUnitStatus.mode.manual OR #statUnitStatus.mode.maintenance;
   #_w10 := #_w9 AND NOT #statPulse[83];   // rising edge
   #statPulse[83] := #_w9;
   #_w11 := NOT #statUnitStatus.mode.production AND "Unit1.Em8.ControlNodes".hipotThickness.sequence.status.inStepIdle AND NOT #statPulse[41];   // rising edge of "Unit1.Em8.ControlNodes".hipotThickness.sequence.status.inStepIdle
   #statPulse[41] := "Unit1.Em8.ControlNodes".hipotThickness.sequence.status.inStepIdle;
   #_w12 := NOT #statUnitStatus.mode.production AND "Unit1.Em8.ControlNodes".GRnR_hipotThickness.sequence.status.inStepIdle AND NOT #statPulse[43];   // rising edge of "Unit1.Em8.ControlNodes".GRnR_hipotThickness.sequence.status.inStepIdle
   #statPulse[43] := "Unit1.Em8.ControlNodes".GRnR_hipotThickness.sequence.status.inStepIdle;
   IF (#_w10 OR #_w11 OR #_w12) AND #statSlmStatus.running AND "Unit1.Em8.HmiInterface".cmThicknessAxisZ.monitoring.axisEnabled THEN
       "Unit1.Em8.ControlNodes".cmThicknessAxisZ.commands.enableAxis := FALSE;
       "Unit1.Em8.HmiInterface".cmThicknessAxisZ.commands.enableAxis := TRUE;
   END_IF;
   IF #statSlmStatus.powerOff OR (#statUnitStatus.state.aborted AND NOT "Unit1.Em8.ControlNodes".cm.brakeTest.thicknessAxisZ.monitoring.busy) OR #statUnitStatus.mode.sleep OR #statUnitStatus.mode.deepsleep OR ("Unit1.EmNodes".safetyStatusZone1.sFDoorOpen AND NOT "Safety.DataFromSafety".gantryTeachMode.auto AND NOT "Safety.DataFromSafety".enableOP.timeExtension AND "Unit1.EmNodes".MobilePanelConnected AND NOT "Unit1.EmNodes".pHmiMode.enable) THEN
       "Unit1.Em8.ControlNodes".cmThicknessAxisZ.commands.enableAxis := FALSE;
       "Unit1.Em8.HmiInterface".cmThicknessAxisZ.commands.enableAxis := FALSE;
   END_IF;
END_REGION

REGION Network 43: PHMI Servo Enable CMs
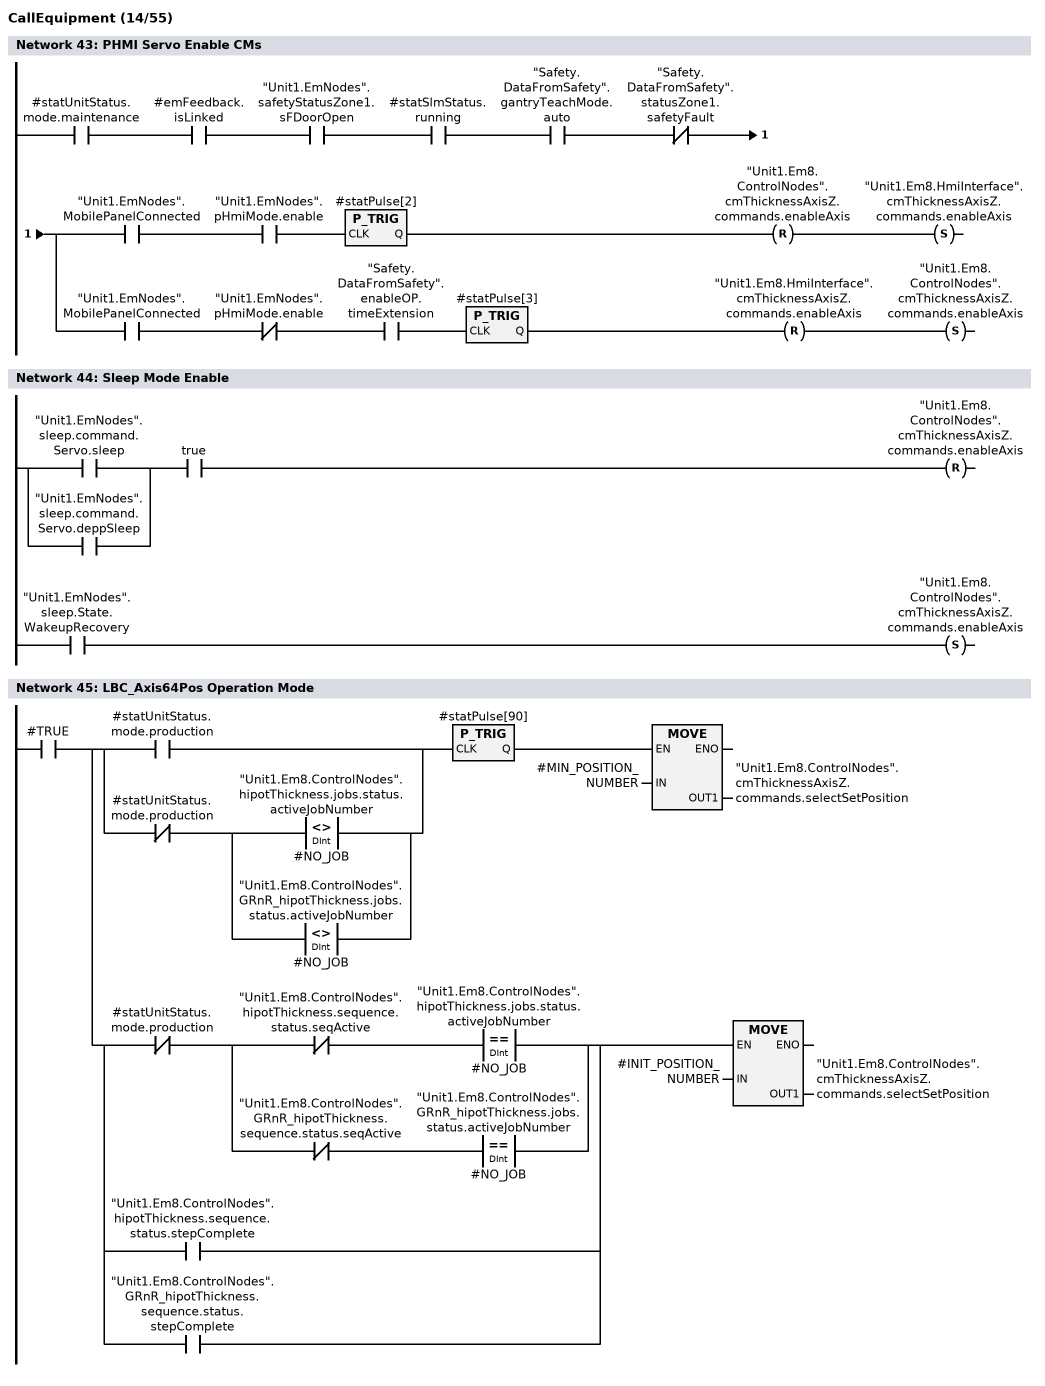
   RUNG wire#powerrail
      Contact( #statUnitStatus.mode.maintenance )
      Contact( #emFeedback.isLinked )
      Contact( "Unit1.EmNodes".safetyStatusZone1.sFDoorOpen )
      Contact( #statSlmStatus.running )
      Contact( "Safety.DataFromSafety".gantryTeachMode.auto )
      I_Contact( "Safety.DataFromSafety".statusZone1.safetyFault )
      wire#w1
      Contact( "Unit1.EmNodes".MobilePanelConnected )
      Contact( "Unit1.EmNodes".pHmiMode.enable )
      P_Trig( #statPulse[2] )
      R_Coil( "Unit1.Em8.ControlNodes".cmThicknessAxisZ.commands.enableAxis )
      S_Coil( "Unit1.Em8.HmiInterface".cmThicknessAxisZ.commands.enableAxis )
   END_RUNG
   RUNG wire#w1
      Contact( "Unit1.EmNodes".MobilePanelConnected )
      I_Contact( "Unit1.EmNodes".pHmiMode.enable )
      Contact( "Safety.DataFromSafety".enableOP.timeExtension )
      P_Trig( #statPulse[3] )
      R_Coil( "Unit1.Em8.HmiInterface".cmThicknessAxisZ.commands.enableAxis )
      S_Coil( "Unit1.Em8.ControlNodes".cmThicknessAxisZ.commands.enableAxis )
   END_RUNG
   // the same network as SCL:
   #_w1 := #statUnitStatus.mode.maintenance AND #emFeedback.isLinked AND "Unit1.EmNodes".safetyStatusZone1.sFDoorOpen AND #statSlmStatus.running AND "Safety.DataFromSafety".gantryTeachMode.auto AND NOT "Safety.DataFromSafety".statusZone1.safetyFault;
   #_w2 := #_w1 AND "Unit1.EmNodes".MobilePanelConnected AND "Unit1.EmNodes".pHmiMode.enable;
   #_w3 := #_w2 AND NOT #statPulse[2];   // rising edge
   #statPulse[2] := #_w2;
   IF #_w3 THEN
       "Unit1.Em8.ControlNodes".cmThicknessAxisZ.commands.enableAxis := FALSE;
       "Unit1.Em8.HmiInterface".cmThicknessAxisZ.commands.enableAxis := TRUE;
   END_IF;
   #_w4 := #_w1 AND "Unit1.EmNodes".MobilePanelConnected AND NOT "Unit1.EmNodes".pHmiMode.enable AND "Safety.DataFromSafety".enableOP.timeExtension;
   #_w5 := #_w4 AND NOT #statPulse[3];   // rising edge
   #statPulse[3] := #_w4;
   IF #_w5 THEN
       "Unit1.Em8.HmiInterface".cmThicknessAxisZ.commands.enableAxis := FALSE;
       "Unit1.Em8.ControlNodes".cmThicknessAxisZ.commands.enableAxis := TRUE;
   END_IF;
END_REGION

REGION Network 44: Sleep Mode Enable
   RUNG wire#powerrail
      Contact( "Unit1.EmNodes".sleep.command.Servo.sleep )
      wire#w1
      Contact( true )
      R_Coil( "Unit1.Em8.ControlNodes".cmThicknessAxisZ.commands.enableAxis )
   END_RUNG
   RUNG wire#powerrail
      Contact( "Unit1.EmNodes".sleep.command.Servo.deppSleep )
   END_RUNG wire#w1
   RUNG wire#powerrail
      Contact( "Unit1.EmNodes".sleep.State.WakeupRecovery )
      S_Coil( "Unit1.Em8.ControlNodes".cmThicknessAxisZ.commands.enableAxis )
   END_RUNG
   // the same network as SCL:
   IF ("Unit1.EmNodes".sleep.command.Servo.sleep OR "Unit1.EmNodes".sleep.command.Servo.deppSleep) AND true THEN
       "Unit1.Em8.ControlNodes".cmThicknessAxisZ.commands.enableAxis := FALSE;
   END_IF;
   IF "Unit1.EmNodes".sleep.State.WakeupRecovery THEN
       "Unit1.Em8.ControlNodes".cmThicknessAxisZ.commands.enableAxis := TRUE;
   END_IF;
END_REGION

REGION Network 45: LBC_Axis64Pos Operation Mode
   RUNG wire#powerrail
      Contact( #TRUE )
      wire#w1
      Contact( #statUnitStatus.mode.production )
      wire#w2
      P_Trig( #statPulse[90] )
      Move(in := #MIN_POSITION_NUMBER, out1 => "Unit1.Em8.ControlNodes".cmThicknessAxisZ.commands.selectSetPosition)
   END_RUNG
   RUNG wire#w1
      I_Contact( #statUnitStatus.mode.production )
      wire#w3
      { S7_Templates := "SrcType := DInt" } NE_Contact(in1 := "Unit1.Em8.ControlNodes".hipotThickness.jobs.status.activeJobNumber, in2 := #NO_JOB)
   END_RUNG wire#w2
   RUNG wire#w3
      { S7_Templates := "SrcType := DInt" } NE_Contact(in1 := "Unit1.Em8.ControlNodes".GRnR_hipotThickness.jobs.status.activeJobNumber, in2 := #NO_JOB)
   END_RUNG wire#w2
   RUNG wire#w1
      I_Contact( #statUnitStatus.mode.production )
      wire#w4
      I_Contact( "Unit1.Em8.ControlNodes".hipotThickness.sequence.status.seqActive )
      { S7_Templates := "SrcType := DInt" } EQ_Contact(in1 := "Unit1.Em8.ControlNodes".hipotThickness.jobs.status.activeJobNumber, in2 := #NO_JOB)
      wire#w5
      Move(in := #INIT_POSITION_NUMBER, out1 => "Unit1.Em8.ControlNodes".cmThicknessAxisZ.commands.selectSetPosition)
   END_RUNG
   RUNG wire#w4
      I_Contact( "Unit1.Em8.ControlNodes".GRnR_hipotThickness.sequence.status.seqActive )
      { S7_Templates := "SrcType := DInt" } EQ_Contact(in1 := "Unit1.Em8.ControlNodes".GRnR_hipotThickness.jobs.status.activeJobNumber, in2 := #NO_JOB)
   END_RUNG wire#w5
   RUNG wire#w1
      Contact( "Unit1.Em8.ControlNodes".hipotThickness.sequence.status.stepComplete )
   END_RUNG wire#w5
   RUNG wire#w1
      Contact( "Unit1.Em8.ControlNodes".GRnR_hipotThickness.sequence.status.stepComplete )
   END_RUNG wire#w5
   // the same network as SCL:
   #_w1 := #TRUE AND (#statUnitStatus.mode.production OR (NOT #statUnitStatus.mode.production AND (("Unit1.Em8.ControlNodes".hipotThickness.jobs.status.activeJobNumber <> #NO_JOB) OR ("Unit1.Em8.ControlNodes".GRnR_hipotThickness.jobs.status.activeJobNumber <> #NO_JOB))));
   #_w2 := #_w1 AND NOT #statPulse[90];   // rising edge
   #statPulse[90] := #_w1;
   IF #_w2 THEN
       "Unit1.Em8.ControlNodes".cmThicknessAxisZ.commands.selectSetPosition := #MIN_POSITION_NUMBER;
   END_IF;
   IF #TRUE AND ((NOT #statUnitStatus.mode.production AND ((NOT "Unit1.Em8.ControlNodes".hipotThickness.sequence.status.seqActive AND ("Unit1.Em8.ControlNodes".hipotThickness.jobs.status.activeJobNumber = #NO_JOB)) OR (NOT "Unit1.Em8.ControlNodes".GRnR_hipotThickness.sequence.status.seqActive AND ("Unit1.Em8.ControlNodes".GRnR_hipotThickness.jobs.status.activeJobNumber = #NO_JOB)))) OR "Unit1.Em8.ControlNodes".hipotThickness.sequence.status.stepComplete OR "Unit1.Em8.ControlNodes".GRnR_hipotThickness.sequence.status.stepComplete) THEN
       "Unit1.Em8.ControlNodes".cmThicknessAxisZ.commands.selectSetPosition := #INIT_POSITION_NUMBER;
   END_IF;
END_REGION

REGION Network 46: Production Mode Change -> Servo Stop
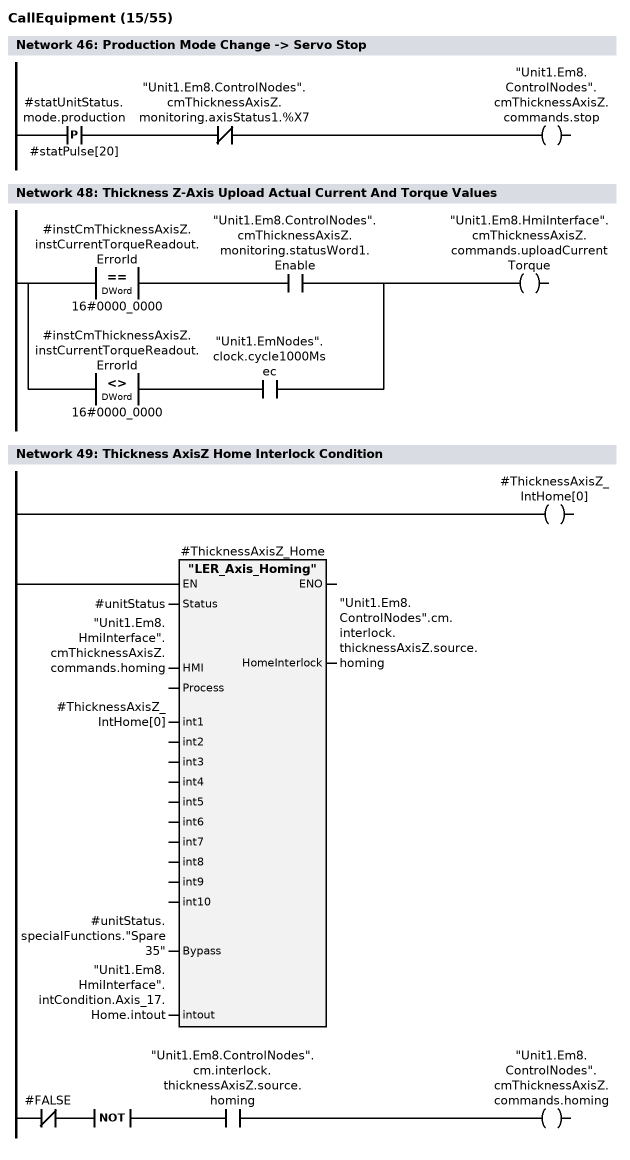
   RUNG wire#powerrail
      P_Contact(operand := #statUnitStatus.mode.production, bit := #statPulse[20])
      I_Contact( "Unit1.Em8.ControlNodes".cmThicknessAxisZ.monitoring.axisStatus1.%X7 )
      Coil( "Unit1.Em8.ControlNodes".cmThicknessAxisZ.commands.stop )
   END_RUNG
   // the same network as SCL:
   #_w1 := #statUnitStatus.mode.production AND NOT #statPulse[20];   // rising edge of #statUnitStatus.mode.production
   #statPulse[20] := #statUnitStatus.mode.production;
   "Unit1.Em8.ControlNodes".cmThicknessAxisZ.commands.stop := #_w1 AND NOT "Unit1.Em8.ControlNodes".cmThicknessAxisZ.monitoring.axisStatus1.%X7;
END_REGION

REGION Network 48: Thickness Z-Axis Upload Actual Current And Torque Values
   RUNG wire#powerrail
      { S7_Templates := "SrcType := DWord" } EQ_Contact(in1 := #instCmThicknessAxisZ.instCurrentTorqueReadout.ErrorId, in2 := 16#0000_0000)
      Contact( "Unit1.Em8.ControlNodes".cmThicknessAxisZ.monitoring.statusWord1.Enable )
      wire#w1
      Coil( "Unit1.Em8.HmiInterface".cmThicknessAxisZ.commands.uploadCurrentTorque )
   END_RUNG
   RUNG wire#powerrail
      { S7_Templates := "SrcType := DWord" } NE_Contact(in1 := #instCmThicknessAxisZ.instCurrentTorqueReadout.ErrorId, in2 := 16#0000_0000)
      Contact( "Unit1.EmNodes".clock.cycle1000Msec )
   END_RUNG wire#w1
   // the same network as SCL:
   "Unit1.Em8.HmiInterface".cmThicknessAxisZ.commands.uploadCurrentTorque := ((#instCmThicknessAxisZ.instCurrentTorqueReadout.ErrorId = 16#0000_0000) AND "Unit1.Em8.ControlNodes".cmThicknessAxisZ.monitoring.statusWord1.Enable) OR ((#instCmThicknessAxisZ.instCurrentTorqueReadout.ErrorId <> 16#0000_0000) AND "Unit1.EmNodes".clock.cycle1000Msec);
END_REGION

REGION Network 49: Thickness AxisZ Home Interlock Condition
   RUNG wire#powerrail
      Coil( #ThicknessAxisZ_IntHome[0] )
   END_RUNG
   RUNG wire#powerrail
      #ThicknessAxisZ_Home(Status := #unitStatus, HMI := "Unit1.Em8.HmiInterface".cmThicknessAxisZ.commands.homing, Process :=, int1 := #ThicknessAxisZ_IntHome[0], int2 :=, int3 :=, int4 :=, int5 :=, int6 :=, int7 :=, int8 :=, int9 :=, int10 :=, Bypass := #unitStatus.specialFunctions."Spare 35", intout := "Unit1.Em8.HmiInterface".intCondition.Axis_17.Home.intout, HomeInterlock => "Unit1.Em8.ControlNodes".cm.interlock.thicknessAxisZ.source.homing)
   END_RUNG
   RUNG wire#powerrail
      I_Contact( #FALSE )
      Not()
      Contact( "Unit1.Em8.ControlNodes".cm.interlock.thicknessAxisZ.source.homing )
      Coil( "Unit1.Em8.ControlNodes".cmThicknessAxisZ.commands.homing )
   END_RUNG
   // the same network as SCL:
   #ThicknessAxisZ_IntHome[0] := TRUE;
   #ThicknessAxisZ_Home(Status := #unitStatus,   // "LER_Axis_Homing"
                        HMI := "Unit1.Em8.HmiInterface".cmThicknessAxisZ.commands.homing,
                        int1 := #ThicknessAxisZ_IntHome[0],
                        Bypass := #unitStatus.specialFunctions."Spare 35",
                        intout := "Unit1.Em8.HmiInterface".intCondition.Axis_17.Home.intout,
                        HomeInterlock => "Unit1.Em8.ControlNodes".cm.interlock.thicknessAxisZ.source.homing);
   "Unit1.Em8.ControlNodes".cmThicknessAxisZ.commands.homing := NOT (NOT #FALSE) AND "Unit1.Em8.ControlNodes".cm.interlock.thicknessAxisZ.source.homing;
END_REGION

REGION Network 50: Thickness AxisZ JOG Interlock Condition
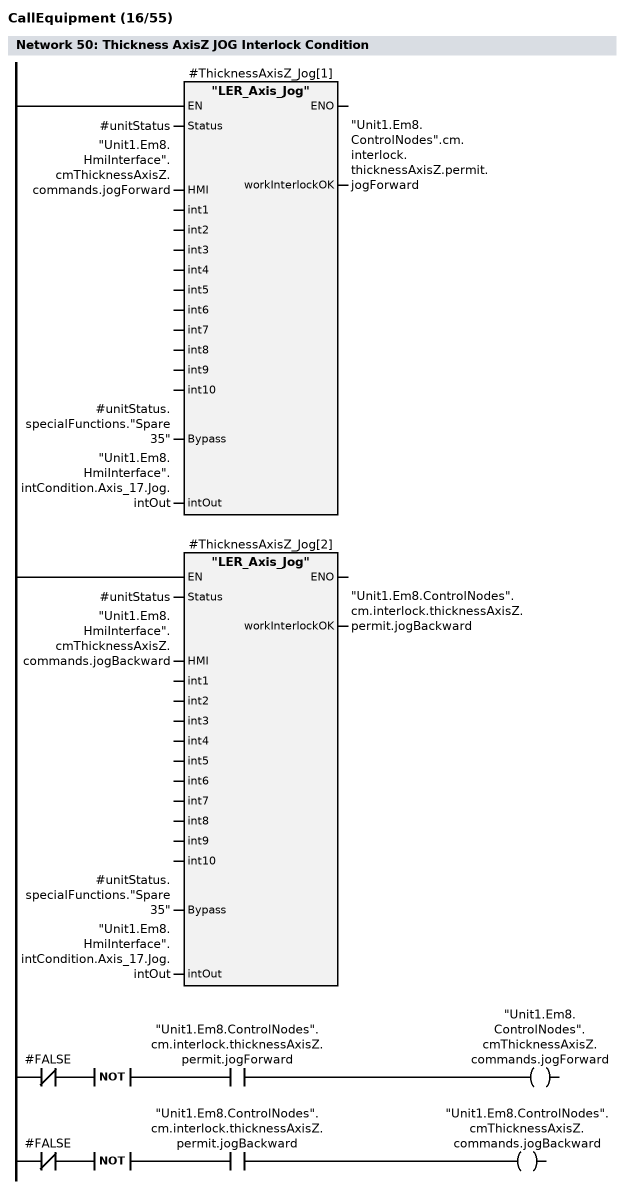
   RUNG wire#powerrail
      #ThicknessAxisZ_Jog[1](Status := #unitStatus, HMI := "Unit1.Em8.HmiInterface".cmThicknessAxisZ.commands.jogForward, int1 :=, int2 :=, int3 :=, int4 :=, int5 :=, int6 :=, int7 :=, int8 :=, int9 :=, int10 :=, Bypass := #unitStatus.specialFunctions."Spare 35", intOut := "Unit1.Em8.HmiInterface".intCondition.Axis_17.Jog.intOut, workInterlockOK => "Unit1.Em8.ControlNodes".cm.interlock.thicknessAxisZ.permit.jogForward)
   END_RUNG
   RUNG wire#powerrail
      #ThicknessAxisZ_Jog[2](Status := #unitStatus, HMI := "Unit1.Em8.HmiInterface".cmThicknessAxisZ.commands.jogBackward, int1 :=, int2 :=, int3 :=, int4 :=, int5 :=, int6 :=, int7 :=, int8 :=, int9 :=, int10 :=, Bypass := #unitStatus.specialFunctions."Spare 35", intOut := "Unit1.Em8.HmiInterface".intCondition.Axis_17.Jog.intOut, workInterlockOK => "Unit1.Em8.ControlNodes".cm.interlock.thicknessAxisZ.permit.jogBackward)
   END_RUNG
   RUNG wire#powerrail
      I_Contact( #FALSE )
      Not()
      Contact( "Unit1.Em8.ControlNodes".cm.interlock.thicknessAxisZ.permit.jogForward )
      Coil( "Unit1.Em8.ControlNodes".cmThicknessAxisZ.commands.jogForward )
   END_RUNG
   RUNG wire#powerrail
      I_Contact( #FALSE )
      Not()
      Contact( "Unit1.Em8.ControlNodes".cm.interlock.thicknessAxisZ.permit.jogBackward )
      Coil( "Unit1.Em8.ControlNodes".cmThicknessAxisZ.commands.jogBackward )
   END_RUNG
   // the same network as SCL:
   #ThicknessAxisZ_Jog[1](Status := #unitStatus,   // "LER_Axis_Jog"
                          HMI := "Unit1.Em8.HmiInterface".cmThicknessAxisZ.commands.jogForward,
                          Bypass := #unitStatus.specialFunctions."Spare 35",
                          intOut := "Unit1.Em8.HmiInterface".intCondition.Axis_17.Jog.intOut,
                          workInterlockOK => "Unit1.Em8.ControlNodes".cm.interlock.thicknessAxisZ.permit.jogForward);
   #ThicknessAxisZ_Jog[2](Status := #unitStatus,   // "LER_Axis_Jog"
                          HMI := "Unit1.Em8.HmiInterface".cmThicknessAxisZ.commands.jogBackward,
                          Bypass := #unitStatus.specialFunctions."Spare 35",
                          intOut := "Unit1.Em8.HmiInterface".intCondition.Axis_17.Jog.intOut,
                          workInterlockOK => "Unit1.Em8.ControlNodes".cm.interlock.thicknessAxisZ.permit.jogBackward);
   "Unit1.Em8.ControlNodes".cmThicknessAxisZ.commands.jogForward := NOT (NOT #FALSE) AND "Unit1.Em8.ControlNodes".cm.interlock.thicknessAxisZ.permit.jogForward;
   "Unit1.Em8.ControlNodes".cmThicknessAxisZ.commands.jogBackward := NOT (NOT #FALSE) AND "Unit1.Em8.ControlNodes".cm.interlock.thicknessAxisZ.permit.jogBackward;
END_REGION

REGION Network 51: Thickness AxisZ Position Absolute Position0
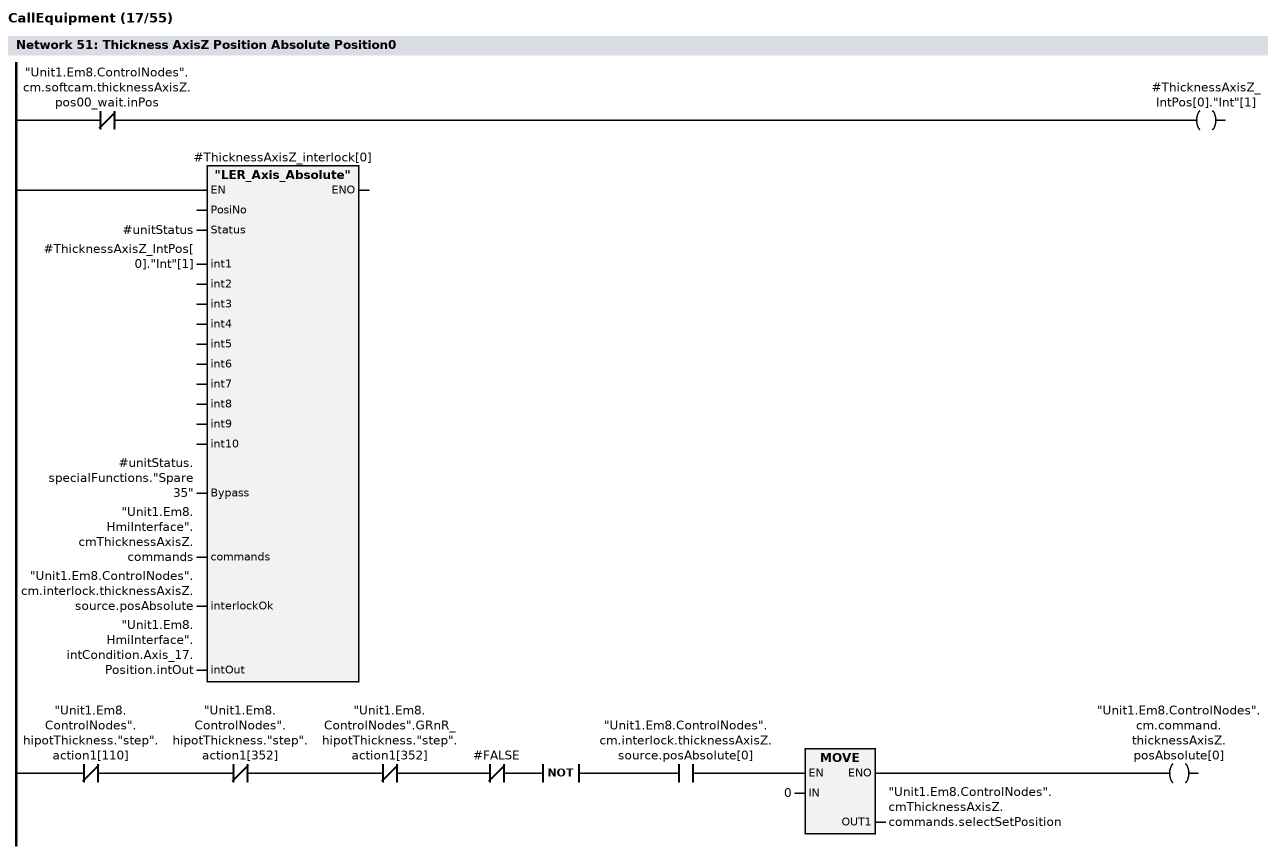
   RUNG wire#powerrail
      I_Contact( "Unit1.Em8.ControlNodes".cm.softcam.thicknessAxisZ.pos00_wait.inPos )
      Coil( #ThicknessAxisZ_IntPos[0]."Int"[1] )
   END_RUNG
   RUNG wire#powerrail
      #ThicknessAxisZ_interlock[0](PosiNo :=, Status := #unitStatus, int1 := #ThicknessAxisZ_IntPos[0]."Int"[1], int2 :=, int3 :=, int4 :=, int5 :=, int6 :=, int7 :=, int8 :=, int9 :=, int10 :=, Bypass := #unitStatus.specialFunctions."Spare 35", commands := "Unit1.Em8.HmiInterface".cmThicknessAxisZ.commands, interlockOk := "Unit1.Em8.ControlNodes".cm.interlock.thicknessAxisZ.source.posAbsolute, intOut := "Unit1.Em8.HmiInterface".intCondition.Axis_17.Position.intOut)
   END_RUNG
   RUNG wire#powerrail
      I_Contact( "Unit1.Em8.ControlNodes".hipotThickness."step".action1[110] )
      I_Contact( "Unit1.Em8.ControlNodes".hipotThickness."step".action1[352] )
      I_Contact( "Unit1.Em8.ControlNodes".GRnR_hipotThickness."step".action1[352] )
      I_Contact( #FALSE )
      Not()
      Contact( "Unit1.Em8.ControlNodes".cm.interlock.thicknessAxisZ.source.posAbsolute[0] )
      Move(in := 0, out1 => "Unit1.Em8.ControlNodes".cmThicknessAxisZ.commands.selectSetPosition)
      Coil( "Unit1.Em8.ControlNodes".cm.command.thicknessAxisZ.posAbsolute[0] )
   END_RUNG
   // the same network as SCL:
   #ThicknessAxisZ_IntPos[0]."Int"[1] := NOT "Unit1.Em8.ControlNodes".cm.softcam.thicknessAxisZ.pos00_wait.inPos;
   #ThicknessAxisZ_interlock[0](Status := #unitStatus,   // "LER_Axis_Absolute"
                           int1 := #ThicknessAxisZ_IntPos[0]."Int"[1],
                           Bypass := #unitStatus.specialFunctions."Spare 35",
                           commands := "Unit1.Em8.HmiInterface".cmThicknessAxisZ.commands,
                           interlockOk := "Unit1.Em8.ControlNodes".cm.interlock.thicknessAxisZ.source.posAbsolute,
                           intOut := "Unit1.Em8.HmiInterface".intCondition.Axis_17.Position.intOut);
   #_w1 := NOT (NOT "Unit1.Em8.ControlNodes".hipotThickness."step".action1[110] AND NOT "Unit1.Em8.ControlNodes".hipotThickness."step".action1[352] AND NOT "Unit1.Em8.ControlNodes".GRnR_hipotThickness."step".action1[352] AND NOT #FALSE) AND "Unit1.Em8.ControlNodes".cm.interlock.thicknessAxisZ.source.posAbsolute[0];
   IF #_w1 THEN "Unit1.Em8.ControlNodes".cmThicknessAxisZ.commands.selectSetPosition := 0; END_IF;
   "Unit1.Em8.ControlNodes".cm.command.thicknessAxisZ.posAbsolute[0] := #_w1;
END_REGION

REGION Network 52: Thickness AxisZ Position Absolute Position1
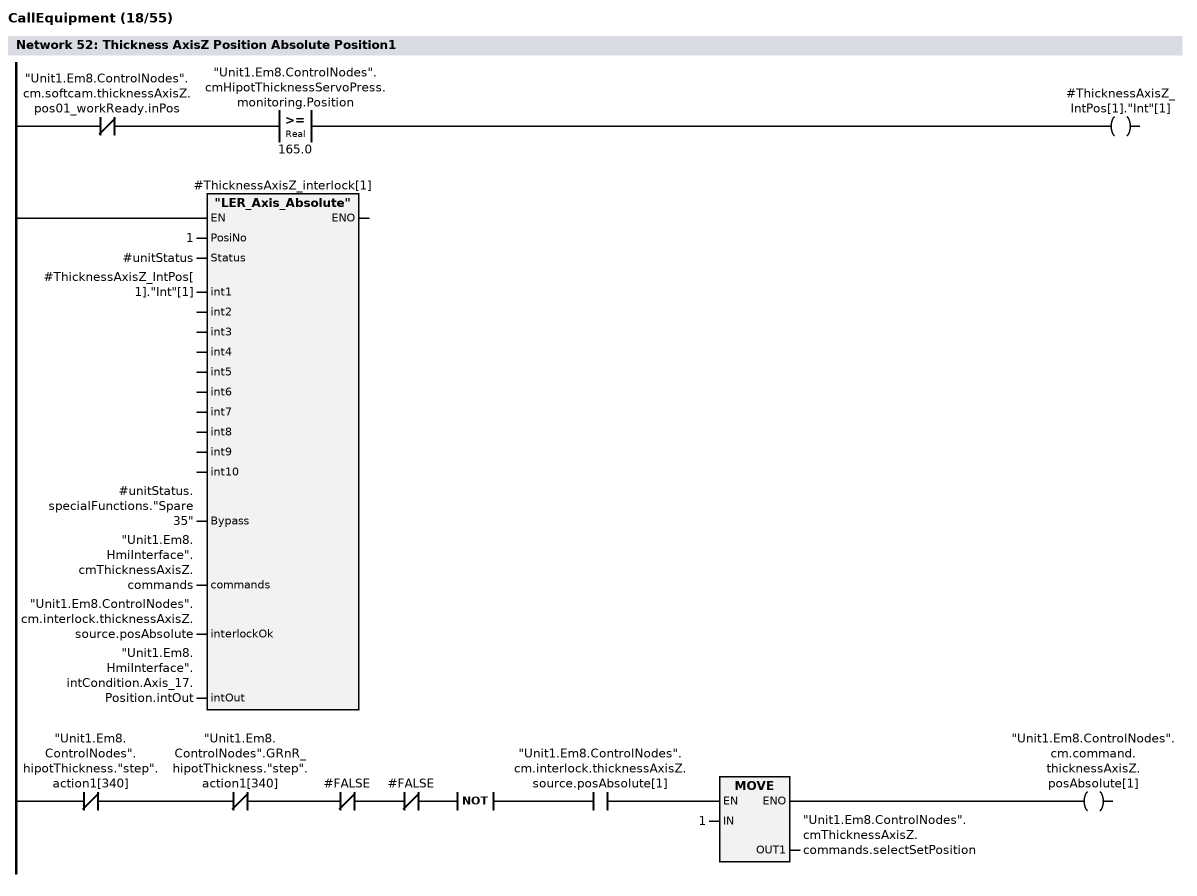
   RUNG wire#powerrail
      I_Contact( "Unit1.Em8.ControlNodes".cm.softcam.thicknessAxisZ.pos01_workReady.inPos )
      { S7_Templates := "SrcType := Real" } GE_Contact(in1 := "Unit1.Em8.ControlNodes".cmHipotThicknessServoPress.monitoring.Position, in2 := 165.0)
      Coil( #ThicknessAxisZ_IntPos[1]."Int"[1] )
   END_RUNG
   RUNG wire#powerrail
      #ThicknessAxisZ_interlock[1](PosiNo := 1, Status := #unitStatus, int1 := #ThicknessAxisZ_IntPos[1]."Int"[1], int2 :=, int3 :=, int4 :=, int5 :=, int6 :=, int7 :=, int8 :=, int9 :=, int10 :=, Bypass := #unitStatus.specialFunctions."Spare 35", commands := "Unit1.Em8.HmiInterface".cmThicknessAxisZ.commands, interlockOk := "Unit1.Em8.ControlNodes".cm.interlock.thicknessAxisZ.source.posAbsolute, intOut := "Unit1.Em8.HmiInterface".intCondition.Axis_17.Position.intOut)
   END_RUNG
   RUNG wire#powerrail
      I_Contact( "Unit1.Em8.ControlNodes".hipotThickness."step".action1[340] )
      I_Contact( "Unit1.Em8.ControlNodes".GRnR_hipotThickness."step".action1[340] )
      I_Contact( #FALSE )
      I_Contact( #FALSE )
      Not()
      Contact( "Unit1.Em8.ControlNodes".cm.interlock.thicknessAxisZ.source.posAbsolute[1] )
      Move(in := 1, out1 => "Unit1.Em8.ControlNodes".cmThicknessAxisZ.commands.selectSetPosition)
      Coil( "Unit1.Em8.ControlNodes".cm.command.thicknessAxisZ.posAbsolute[1] )
   END_RUNG
   // the same network as SCL:
   #ThicknessAxisZ_IntPos[1]."Int"[1] := NOT "Unit1.Em8.ControlNodes".cm.softcam.thicknessAxisZ.pos01_workReady.inPos AND ("Unit1.Em8.ControlNodes".cmHipotThicknessServoPress.monitoring.Position >= 165.0);
   #ThicknessAxisZ_interlock[1](PosiNo := 1,   // "LER_Axis_Absolute"
                           Status := #unitStatus,
                           int1 := #ThicknessAxisZ_IntPos[1]."Int"[1],
                           Bypass := #unitStatus.specialFunctions."Spare 35",
                           commands := "Unit1.Em8.HmiInterface".cmThicknessAxisZ.commands,
                           interlockOk := "Unit1.Em8.ControlNodes".cm.interlock.thicknessAxisZ.source.posAbsolute,
                           intOut := "Unit1.Em8.HmiInterface".intCondition.Axis_17.Position.intOut);
   #_w1 := NOT (NOT "Unit1.Em8.ControlNodes".hipotThickness."step".action1[340] AND NOT "Unit1.Em8.ControlNodes".GRnR_hipotThickness."step".action1[340] AND NOT #FALSE AND NOT #FALSE) AND "Unit1.Em8.ControlNodes".cm.interlock.thicknessAxisZ.source.posAbsolute[1];
   IF #_w1 THEN "Unit1.Em8.ControlNodes".cmThicknessAxisZ.commands.selectSetPosition := 1; END_IF;
   "Unit1.Em8.ControlNodes".cm.command.thicknessAxisZ.posAbsolute[1] := #_w1;
END_REGION

